LIN {X 0,Y 573.234,Z 422.71,A -85,B 0,C 180,E1 -2362.338,E2 -2362.338} C_VEL
LIN {X 0,Y 573.247,Z 422.704,A -85,B 0,C 180,E1 -2364.401,E2 -2364.401} C_VEL
LIN {X 0,Y 572.62,Z 422.786,A -85,B 0,C 180,E1 -2364.987,E2 -2364.987} C_VEL
LIN {X 0,Y 569.776,Z 423.137,A -85,B 0,C 180,E1 -2365.938,E2 -2365.938} C_VEL
LIN {X 0,Y 567.346,Z 423.44,A -85,B 0,C 180,E1 -2366.704,E2 -2366.704} C_VEL
LIN {X 0,Y 566.295,Z 423.569,A -85,B 0,C 180,E1 -2367.295,E2 -2367.295} C_VEL
LIN {X 0,Y 566.207,Z 423.58,A -85,B 0,C 180,E1 -2367.495,E2 -2367.495} C_VEL
LIN {X 0,Y 566.184,Z 423.588,A -85,B 0,C 180,E1 -2370.593,E2 -2370.593} C_VEL
LIN {X 0,Y 566.225,Z 423.58,A -85,B 0,C 180,E1 -2373.102,E2 -2373.102} C_VEL
LIN {X 0,Y 566.212,Z 423.583,A -85,B 0,C 180,E1 -2376.217,E2 -2376.217} C_VEL
LIN {X 0,Y 566.212,Z 423.58,A -85,B 0,C 180,E1 -2379.274,E2 -2379.274} C_VEL
LIN {X 0,Y 566.215,Z 423.58,A -85,B 0,C 180,E1 -2382.088,E2 -2382.088} C_VEL
LIN {X 0,Y 566.172,Z 423.584,A -85,B 0,C 180,E1 -2385.036,E2 -2385.036} C_VEL
LIN {X 0,Y 566.189,Z 423.583,A -85,B 0,C 180,E1 -2387.911,E2 -2387.911} C_VEL
LIN {X 0,Y 566.222,Z 423.579,A -85,B 0,C 180,E1 -2390.728,E2 -2390.728} C_VEL
LIN {X 0,Y 566.219,Z 423.582,A -85,B 0,C 180,E1 -2393.784,E2 -2393.784} C_VEL
LIN {X 0,Y 566.213,Z 423.581,A -85,B 0,C 180,E1 -2396.266,E2 -2396.266} C_VEL
LIN {X 0,Y 566.195,Z 423.582,A -85,B 0,C 180,E1 -2398.924,E2 -2398.924} C_VEL
LIN {X 0,Y 566.196,Z 423.584,A -85,B 0,C 180,E1 -2401.047,E2 -2401.047} C_VEL
LIN {X 0,Y 566.219,Z 423.582,A -85,B 0,C 180,E1 -2403.46,E2 -2403.46} C_VEL
LIN {X 0,Y 566.201,Z 423.582,A -85,B 0,C 180,E1 -2405.82,E2 -2405.82} C_VEL
LIN {X 0,Y 566.211,Z 423.583,A -85,B 0,C 180,E1 -2408.903,E2 -2408.903} C_VEL
LIN {X 0,Y 566.203,Z 423.581,A -85,B 0,C 180,E1 -2411.173,E2 -2411.173} C_VEL
LIN {X 0,Y 566.217,Z 423.582,A -85,B 0,C 180,E1 -2413.413,E2 -2413.413} C_VEL
LIN {X 0,Y 566.201,Z 423.581,A -85,B 0,C 180,E1 -2416.359,E2 -2416.359} C_VEL
LIN {X 0,Y 566.239,Z 423.58,A -85,B 0,C 180,E1 -2418.676,E2 -2418.676} C_VEL
LIN {X 0,Y 566.232,Z 423.582,A -85,B 0,C 180,E1 -2421.435,E2 -2421.435} C_VEL
LIN {X 0,Y 566.259,Z 423.577,A -85,B 0,C 180,E1 -2424.302,E2 -2424.302} C_VEL
LIN {X 0,Y 566.287,Z 423.572,A -85,B 0,C 180,E1 -2427.866,E2 -2427.866} C_VEL
LIN {X 0,Y 566.302,Z 423.569,A -85,B 0,C 180,E1 -2430.711,E2 -2430.711} C_VEL
LIN {X 0,Y 566.274,Z 423.573,A -85,B 0,C 180,E1 -2432.845,E2 -2432.845} C_VEL
LIN {X 0,Y 566.266,Z 423.573,A -85,B 0,C 180,E1 -2435.698,E2 -2435.698} C_VEL
LIN {X 0,Y 566.211,Z 423.58,A -85,B 0,C 180,E1 -2438.566,E2 -2438.566} C_VEL
LIN {X 0,Y 566.246,Z 423.576,A -85,B 0,C 180,E1 -2441.454,E2 -2441.454} C_VEL
LIN {X 0,Y 566.239,Z 423.578,A -85,B 0,C 180,E1 -2444.506,E2 -2444.506} C_VEL
LIN {X 0,Y 566.202,Z 423.584,A -85,B 0,C 180,E1 -2447.331,E2 -2447.331} C_VEL
LIN {X 0,Y 566.211,Z 423.584,A -85,B 0,C 180,E1 -2450.337,E2 -2450.337} C_VEL
LIN {X 0,Y 566.193,Z 423.583,A -85,B 0,C 180,E1 -2453.403,E2 -2453.403} C_VEL
LIN {X 0,Y 566.217,Z 423.583,A -85,B 0,C 180,E1 -2455.748,E2 -2455.748} C_VEL
LIN {X 0,Y 566.209,Z 423.581,A -85,B 0,C 180,E1 -2458.202,E2 -2458.202} C_VEL
LIN {X 0,Y 566.201,Z 423.584,A -85,B 0,C 180,E1 -2461.077,E2 -2461.077} C_VEL
LIN {X 0,Y 566.188,Z 423.585,A -85,B 0,C 180,E1 -2463.73,E2 -2463.73} C_VEL
LIN {X 0,Y 565.994,Z 423.636,A -85,B 0,C 180,E1 -2465.704,E2 -2465.704} C_VEL
LIN {X 0,Y 565.976,Z 426.477,A -85,B 0,C 180,E1 -2468.528,E2 -2468.528} C_VEL
LIN {X 0,Y 565.936,Z 429.152,A -85,B 0,C 180,E1 -2471.16,E2 -2471.16} C_VEL
LIN {X 0,Y 565.954,Z 432.13,A -85,B 0,C 180,E1 -2474.059,E2 -2474.059} C_VEL
LIN {X 0,Y 565.928,Z 435.2,A -85,B 0,C 180,E1 -2477.112,E2 -2477.112} C_VEL
LIN {X 0,Y 565.889,Z 438.183,A -85,B 0,C 180,E1 -2479.773,E2 -2479.773} C_VEL
LIN {X 0,Y 565.844,Z 441.501,A -85,B 0,C 180,E1 -2482.645,E2 -2482.645} C_VEL
LIN {X 0,Y 565.859,Z 444.449,A -85,B 0,C 180,E1 -2485.157,E2 -2485.157} C_VEL
LIN {X 0,Y 565.879,Z 446.388,A -85,B 0,C 180,E1 -2486.791,E2 -2486.791} C_VEL
LIN {X 0,Y 567.394,Z 454.471,A -85,B 0,C 180,E1 -2486.992,E2 -2486.992} C_VEL
LIN {X 0,Y 567.255,Z 468.399,A -85,B 0,C 180,E1 -2487.361,E2 -2487.361} C_VEL
LIN {X 0,Y 567.079,Z 481.532,A -85,B 0,C 180,E1 -2487.85,E2 -2487.85} C_VEL
LIN {X 0,Y 566.886,Z 495.141,A -85,B 0,C 180,E1 -2488.517,E2 -2488.517} C_VEL
LIN {X 0,Y 566.716,Z 507.038,A -85,B 0,C 180,E1 -2489.251,E2 -2489.251} C_VEL
LIN {X 0,Y 566.534,Z 518.876,A -85,B 0,C 180,E1 -2490.148,E2 -2490.148} C_VEL
LIN {X 0,Y 566.38,Z 528.827,A -85,B 0,C 180,E1 -2491.057,E2 -2491.057} C_VEL
LIN {X 0,Y 566.217,Z 538.024,A -85,B 0,C 180,E1 -2492.059,E2 -2492.059} C_VEL
LIN {X 0,Y 566.123,Z 547.123,A -85,B 0,C 180,E1 -2493.256,E2 -2493.256} C_VEL
LIN {X 0,Y 566.004,Z 554.487,A -85,B 0,C 180,E1 -2494.438,E2 -2494.438} C_VEL
LIN {X 0,Y 565.951,Z 561.337,A -85,B 0,C 180,E1 -2495.808,E2 -2495.808} C_VEL
LIN {X 0,Y 565.93,Z 565.213,A -85,B 0,C 180,E1 -2496.773,E2 -2496.773} C_VEL
LIN {X 0,Y 565.88,Z 569.42,A -85,B 0,C 180,E1 -2498.124,E2 -2498.124} C_VEL
LIN {X 0,Y 565.891,Z 571.213,A -85,B 0,C 180,E1 -2498.89,E2 -2498.89} C_VEL
LIN {X 0,Y 565.832,Z 573.597,A -85,B 0,C 180,E1 -2500.406,E2 -2500.406} C_VEL
LIN {X 0,Y 565.83,Z 574.477,A -85,B 0,C 180,E1 -2501.909,E2 -2501.909} C_VEL
LIN {X 0,Y 565.841,Z 573.9,A -85,B 0,C 180,E1 -2503.401,E2 -2503.401} C_VEL
LIN {X 0,Y 565.84,Z 571.856,A -85,B 0,C 180,E1 -2504.88,E2 -2504.88} C_VEL
LIN {X 0,Y 565.899,Z 568.345,A -85,B 0,C 180,E1 -2506.351,E2 -2506.351} C_VEL
LIN {X 0,Y 565.941,Z 563.307,A -85,B 0,C 180,E1 -2507.812,E2 -2507.812} C_VEL
LIN {X 0,Y 565.973,Z 558.307,A -85,B 0,C 180,E1 -2508.93,E2 -2508.93} C_VEL
LIN {X 0,Y 566.075,Z 551.435,A -85,B 0,C 180,E1 -2510.171,E2 -2510.171} C_VEL
LIN {X 0,Y 566.125,Z 542.804,A -85,B 0,C 180,E1 -2511.433,E2 -2511.433} C_VEL
LIN {X 0,Y 566.313,Z 533.799,A -85,B 0,C 180,E1 -2512.513,E2 -2512.513} C_VEL
LIN {X 0,Y 566.448,Z 522.985,A -85,B 0,C 180,E1 -2513.589,E2 -2513.589} C_VEL
LIN {X 0,Y 566.645,Z 512.043,A -85,B 0,C 180,E1 -2514.484,E2 -2514.484} C_VEL
LIN {X 0,Y 566.779,Z 500.105,A -85,B 0,C 180,E1 -2515.288,E2 -2515.288} C_VEL
LIN {X 0,Y 567.003,Z 486.787,A -85,B 0,C 180,E1 -2516.002,E2 -2516.002} C_VEL
LIN {X 0,Y 567.196,Z 473.978,A -85,B 0,C 180,E1 -2516.537,E2 -2516.537} C_VEL
LIN {X 0,Y 567.341,Z 460.316,A -85,B 0,C 180,E1 -2516.96,E2 -2516.96} C_VEL
LIN {X 0,Y 567.167,Z 452.884,A -85,B 0,C 180,E1 -2517.137,E2 -2517.137} C_VEL
LIN {X 0,Y 565.851,Z 446.378,A -85,B 0,C 180,E1 -2517.308,E2 -2517.308} C_VEL
LIN {X 0,Y 565.889,Z 443.19,A -85,B 0,C 180,E1 -2520,E2 -2520} C_VEL
LIN {X 0,Y 565.883,Z 439.872,A -85,B 0,C 180,E1 -2522.847,E2 -2522.847} C_VEL
LIN {X 0,Y 565.959,Z 436.605,A -85,B 0,C 180,E1 -2525.701,E2 -2525.701} C_VEL
LIN {X 0,Y 565.979,Z 434.458,A -85,B 0,C 180,E1 -2527.851,E2 -2527.851} C_VEL
LIN {X 0,Y 566.06,Z 431.516,A -85,B 0,C 180,E1 -2531.241,E2 -2531.241} C_VEL
LIN {X 0,Y 566.065,Z 428.336,A -85,B 0,C 180,E1 -2534.443,E2 -2534.443} C_VEL
LIN {X 0,Y 566.096,Z 425.665,A -85,B 0,C 180,E1 -2537.335,E2 -2537.335} C_VEL
LIN {X 0,Y 566.111,Z 423.597,A -85,B 0,C 180,E1 -2539.584,E2 -2539.584} C_VEL
LIN {X 0,Y 566.191,Z 423.584,A -85,B 0,C 180,E1 -2541.863,E2 -2541.863} C_VEL
LIN {X 0,Y 566.229,Z 423.575,A -85,B 0,C 180,E1 -2544.961,E2 -2544.961} C_VEL
LIN {X 0,Y 566.219,Z 423.576,A -85,B 0,C 180,E1 -2547.339,E2 -2547.339} C_VEL
LIN {X 0,Y 566.222,Z 423.58,A -85,B 0,C 180,E1 -2549.768,E2 -2549.768} C_VEL
LIN {X 0,Y 566.204,Z 423.581,A -85,B 0,C 180,E1 -2552.431,E2 -2552.431} C_VEL
LIN {X 0,Y 566.208,Z 423.577,A -85,B 0,C 180,E1 -2554.995,E2 -2554.995} C_VEL
LIN {X 0,Y 566.192,Z 423.581,A -85,B 0,C 180,E1 -2557.461,E2 -2557.461} C_VEL
LIN {X 0,Y 566.223,Z 423.581,A -85,B 0,C 180,E1 -2560.198,E2 -2560.198} C_VEL
LIN {X 0,Y 566.202,Z 423.579,A -85,B 0,C 180,E1 -2563.054,E2 -2563.054} C_VEL
LIN {X 0,Y 566.199,Z 423.587,A -85,B 0,C 180,E1 -2566.049,E2 -2566.049} C_VEL
LIN {X 0,Y 566.209,Z 423.582,A -85,B 0,C 180,E1 -2568.864,E2 -2568.864} C_VEL
LIN {X 0,Y 566.262,Z 423.679,A -85,B 0,C 180,E1 -2569.587,E2 -2569.587} C_VEL
LIN {X 0,Y 566.891,Z 427.712,A -85,B 0,C 180,E1 -2571.356,E2 -2571.356} C_VEL
LIN {X 0,Y 566.768,Z 433.908,A -85,B 0,C 180,E1 -2573.708,E2 -2573.708} C_VEL
LIN {X 0,Y 566.619,Z 441.021,A -85,B 0,C 180,E1 -2576.204,E2 -2576.204} C_VEL
LIN {X 0,Y 566.57,Z 449.293,A -85,B 0,C 180,E1 -2578.86,E2 -2578.86} C_VEL
LIN {X 0,Y 566.478,Z 459.198,A -85,B 0,C 180,E1 -2581.872,E2 -2581.872} C_VEL
LIN {X 0,Y 566.392,Z 468.297,A -85,B 0,C 180,E1 -2584.639,E2 -2584.639} C_VEL
LIN {X 0,Y 566.27,Z 477.307,A -85,B 0,C 180,E1 -2587.373,E2 -2587.373} C_VEL
LIN {X 0,Y 566.193,Z 487.546,A -85,B 0,C 180,E1 -2590.419,E2 -2590.419} C_VEL
LIN {X 0,Y 566.11,Z 497.786,A -85,B 0,C 180,E1 -2593.41,E2 -2593.41} C_VEL
LIN {X 0,Y 566.085,Z 502.186,A -85,B 0,C 180,E1 -2594.68,E2 -2594.68} C_VEL
LIN {X 0,Y 567.44,Z 510.182,A -85,B 0,C 180,E1 -2594.861,E2 -2594.861} C_VEL
LIN {X 0,Y 567.305,Z 524.025,A -85,B 0,C 180,E1 -2595.185,E2 -2595.185} C_VEL
LIN {X 0,Y 567.112,Z 537.717,A -85,B 0,C 180,E1 -2595.65,E2 -2595.65} C_VEL
LIN {X 0,Y 566.975,Z 551.647,A -85,B 0,C 180,E1 -2596.287,E2 -2596.287} C_VEL
LIN {X 0,Y 566.763,Z 564.104,A -85,B 0,C 180,E1 -2597.012,E2 -2597.012} C_VEL
LIN {X 0,Y 566.576,Z 576.643,A -85,B 0,C 180,E1 -2597.918,E2 -2597.918} C_VEL
LIN {X 0,Y 566.446,Z 587.32,A -85,B 0,C 180,E1 -2598.861,E2 -2598.861} C_VEL
LIN {X 0,Y 566.206,Z 597.853,A -85,B 0,C 180,E1 -2599.993,E2 -2599.993} C_VEL
LIN {X 0,Y 566.132,Z 606.173,A -85,B 0,C 180,E1 -2601.073,E2 -2601.073} C_VEL
LIN {X 0,Y 566.046,Z 614.128,A -85,B 0,C 180,E1 -2602.33,E2 -2602.33} C_VEL
LIN {X 0,Y 565.943,Z 620.528,A -85,B 0,C 180,E1 -2603.583,E2 -2603.583} C_VEL
LIN {X 0,Y 565.928,Z 624.961,A -85,B 0,C 180,E1 -2604.656,E2 -2604.656} C_VEL
LIN {X 0,Y 565.956,Z 628.443,A -85,B 0,C 180,E1 -2605.727,E2 -2605.727} C_VEL
LIN {X 0,Y 565.874,Z 631.832,A -85,B 0,C 180,E1 -2607.152,E2 -2607.152} C_VEL
LIN {X 0,Y 565.84,Z 633.833,A -85,B 0,C 180,E1 -2608.577,E2 -2608.577} C_VEL
LIN {X 0,Y 565.837,Z 634.5,A -85,B 0,C 180,E1 -2610,E2 -2610} C_VEL
LIN {X 0,Y 565.84,Z 633.833,A -85,B 0,C 180,E1 -2611.423,E2 -2611.423} C_VEL
LIN {X 0,Y 565.874,Z 631.834,A -85,B 0,C 180,E1 -2612.848,E2 -2612.848} C_VEL
LIN {X 0,Y 565.956,Z 628.445,A -85,B 0,C 180,E1 -2614.273,E2 -2614.273} C_VEL
LIN {X 0,Y 565.988,Z 623.568,A -85,B 0,C 180,E1 -2615.701,E2 -2615.701} C_VEL
LIN {X 0,Y 565.992,Z 619.045,A -85,B 0,C 180,E1 -2616.739,E2 -2616.739} C_VEL
LIN {X 0,Y 566.047,Z 612.038,A -85,B 0,C 180,E1 -2618.029,E2 -2618.029} C_VEL
LIN {X 0,Y 566.177,Z 603.56,A -85,B 0,C 180,E1 -2619.286,E2 -2619.286} C_VEL
LIN {X 0,Y 566.294,Z 594.709,A -85,B 0,C 180,E1 -2620.367,E2 -2620.367} C_VEL
LIN {X 0,Y 566.485,Z 583.993,A -85,B 0,C 180,E1 -2621.449,E2 -2621.449} C_VEL
LIN {X 0,Y 566.638,Z 573.145,A -85,B 0,C 180,E1 -2622.354,E2 -2622.354} C_VEL
LIN {X 0,Y 566.774,Z 561.262,A -85,B 0,C 180,E1 -2623.17,E2 -2623.17} C_VEL
LIN {X 0,Y 567.046,Z 548.1,A -85,B 0,C 180,E1 -2623.894,E2 -2623.894} C_VEL
LIN {X 0,Y 567.194,Z 535.146,A -85,B 0,C 180,E1 -2624.45,E2 -2624.45} C_VEL
LIN {X 0,Y 567.335,Z 520.935,A -85,B 0,C 180,E1 -2624.899,E2 -2624.899} C_VEL
LIN {X 0,Y 567.341,Z 508.652,A -85,B 0,C 180,E1 -2625.17,E2 -2625.17} C_VEL
LIN {X 0,Y 566.086,Z 502.186,A -85,B 0,C 180,E1 -2625.32,E2 -2625.32} C_VEL
LIN {X 0,Y 566.15,Z 492.666,A -85,B 0,C 180,E1 -2628.079,E2 -2628.079} C_VEL
LIN {X 0,Y 566.215,Z 483.706,A -85,B 0,C 180,E1 -2630.716,E2 -2630.716} C_VEL
LIN {X 0,Y 566.312,Z 474.747,A -85,B 0,C 180,E1 -2633.398,E2 -2633.398} C_VEL
LIN {X 0,Y 566.406,Z 465.778,A -85,B 0,C 180,E1 -2636.134,E2 -2636.134} C_VEL
LIN {X 0,Y 566.502,Z 456.675,A -85,B 0,C 180,E1 -2638.935,E2 -2638.935} C_VEL
LIN {X 0,Y 566.607,Z 447.555,A -85,B 0,C 180,E1 -2641.813,E2 -2641.813} C_VEL
LIN {X 0,Y 566.777,Z 438.577,A -85,B 0,C 180,E1 -2644.777,E2 -2644.777} C_VEL
LIN {X 0,Y 566.892,Z 430.796,A -85,B 0,C 180,E1 -2647.492,E2 -2647.492} C_VEL
LIN {X 0,Y 566.907,Z 427.604,A -85,B 0,C 180,E1 -2648.646,E2 -2648.646} C_VEL
LIN {X 0,Y 566.223,Z 423.582,A -85,B 0,C 180,E1 -2650.252,E2 -2650.252} C_VEL
LIN {X 0,Y 566.198,Z 423.583,A -85,B 0,C 180,E1 -2653.053,E2 -2653.053} C_VEL
LIN {X 0,Y 566.199,Z 423.583,A -85,B 0,C 180,E1 -2656.048,E2 -2656.048} C_VEL
LIN {X 0,Y 566.208,Z 423.582,A -85,B 0,C 180,E1 -2658.863,E2 -2658.863} C_VEL
LIN {X 0,Y 566.186,Z 423.586,A -85,B 0,C 180,E1 -2661.637,E2 -2661.637} C_VEL
LIN {X 0,Y 566.191,Z 423.584,A -85,B 0,C 180,E1 -2664.31,E2 -2664.31} C_VEL
LIN {X 0,Y 566.224,Z 423.579,A -85,B 0,C 180,E1 -2666.898,E2 -2666.898} C_VEL
LIN {X 0,Y 566.189,Z 423.583,A -85,B 0,C 180,E1 -2669.408,E2 -2669.408} C_VEL
LIN {X 0,Y 566.222,Z 423.579,A -85,B 0,C 180,E1 -2671.858,E2 -2671.858} C_VEL
LIN {X 0,Y 566.222,Z 423.583,A -85,B 0,C 180,E1 -2674.251,E2 -2674.251} C_VEL
LIN {X 0,Y 566.185,Z 423.585,A -85,B 0,C 180,E1 -2676.713,E2 -2676.713} C_VEL
LIN {X 0,Y 566.214,Z 423.584,A -85,B 0,C 180,E1 -2679.663,E2 -2679.663} C_VEL
LIN {X 0,Y 566.198,Z 423.585,A -85,B 0,C 180,E1 -2682.668,E2 -2682.668} C_VEL
LIN {X 0,Y 566.227,Z 423.579,A -85,B 0,C 180,E1 -2685.627,E2 -2685.627} C_VEL
LIN {X 0,Y 566.268,Z 423.573,A -85,B 0,C 180,E1 -2688.654,E2 -2688.654} C_VEL
LIN {X 0,Y 566.243,Z 423.576,A -85,B 0,C 180,E1 -2691.435,E2 -2691.435} C_VEL
LIN {X 0,Y 566.257,Z 423.575,A -85,B 0,C 180,E1 -2694.302,E2 -2694.302} C_VEL
LIN {X 0,Y 566.275,Z 423.574,A -85,B 0,C 180,E1 -2697.866,E2 -2697.866} C_VEL
LIN {X 0,Y 566.299,Z 423.57,A -85,B 0,C 180,E1 -2700.711,E2 -2700.711} C_VEL
LIN {X 0,Y 566.274,Z 423.574,A -85,B 0,C 180,E1 -2702.846,E2 -2702.846} C_VEL
LIN {X 0,Y 566.266,Z 423.576,A -85,B 0,C 180,E1 -2705.698,E2 -2705.698} C_VEL
LIN {X 0,Y 566.242,Z 423.581,A -85,B 0,C 180,E1 -2708.566,E2 -2708.566} C_VEL
LIN {X 0,Y 566.235,Z 423.581,A -85,B 0,C 180,E1 -2711.455,E2 -2711.455} C_VEL
LIN {X 0,Y 566.227,Z 423.579,A -85,B 0,C 180,E1 -2714.507,E2 -2714.507} C_VEL
LIN {X 0,Y 566.199,Z 423.582,A -85,B 0,C 180,E1 -2717.332,E2 -2717.332} C_VEL
LIN {X 0,Y 566.215,Z 423.58,A -85,B 0,C 180,E1 -2720.337,E2 -2720.337} C_VEL
LIN {X 0,Y 566.185,Z 423.585,A -85,B 0,C 180,E1 -2723.404,E2 -2723.404} C_VEL
LIN {X 0,Y 566.21,Z 423.58,A -85,B 0,C 180,E1 -2725.749,E2 -2725.749} C_VEL
LIN {X 0,Y 566.207,Z 423.58,A -85,B 0,C 180,E1 -2727.495,E2 -2727.495} C_VEL
LIN {X 0,Y 565.531,Z 423.667,A -85,B 0,C 180,E1 -2728.089,E2 -2728.089} C_VEL
LIN {X 0,Y 562.662,Z 424.025,A -85,B 0,C 180,E1 -2729.052,E2 -2729.052} C_VEL
LIN {X 0,Y 560.248,Z 424.324,A -85,B 0,C 180,E1 -2729.828,E2 -2729.828} C_VEL
LIN {X 0,Y 559.22,Z 424.454,A -85,B 0,C 180,E1 -2730.427,E2 -2730.427} C_VEL
LIN {X 0,Y 559.141,Z 424.459,A -85,B 0,C 180,E1 -2730.629,E2 -2730.629} C_VEL
LIN {X 0,Y 559.161,Z 424.461,A -85,B 0,C 180,E1 -2733.575,E2 -2733.575} C_VEL
LIN {X 0,Y 559.164,Z 424.459,A -85,B 0,C 180,E1 -2736.449,E2 -2736.449} C_VEL
LIN {X 0,Y 559.172,Z 424.46,A -85,B 0,C 180,E1 -2738.935,E2 -2738.935} C_VEL
LIN {X 0,Y 559.178,Z 424.457,A -85,B 0,C 180,E1 -2742.138,E2 -2742.138} C_VEL
LIN {X 0,Y 559.139,Z 424.461,A -85,B 0,C 180,E1 -2744.74,E2 -2744.74} C_VEL
LIN {X 0,Y 559.159,Z 424.462,A -85,B 0,C 180,E1 -2747.257,E2 -2747.257} C_VEL
LIN {X 0,Y 559.185,Z 424.457,A -85,B 0,C 180,E1 -2750.136,E2 -2750.136} C_VEL
LIN {X 0,Y 559.147,Z 424.461,A -85,B 0,C 180,E1 -2752.893,E2 -2752.893} C_VEL
LIN {X 0,Y 559.159,Z 424.461,A -85,B 0,C 180,E1 -2755.557,E2 -2755.557} C_VEL
LIN {X 0,Y 559.167,Z 424.461,A -85,B 0,C 180,E1 -2758.138,E2 -2758.138} C_VEL
LIN {X 0,Y 559.159,Z 424.462,A -85,B 0,C 180,E1 -2760.648,E2 -2760.648} C_VEL
LIN {X 0,Y 559.173,Z 424.457,A -85,B 0,C 180,E1 -2763.173,E2 -2763.173} C_VEL
LIN {X 0,Y 559.159,Z 424.459,A -85,B 0,C 180,E1 -2765.495,E2 -2765.495} C_VEL
LIN {X 0,Y 559.175,Z 424.457,A -85,B 0,C 180,E1 -2768.624,E2 -2768.624} C_VEL
LIN {X 0,Y 559.166,Z 424.458,A -85,B 0,C 180,E1 -2770.927,E2 -2770.927} C_VEL
LIN {X 0,Y 559.169,Z 424.458,A -85,B 0,C 180,E1 -2773.948,E2 -2773.948} C_VEL
LIN {X 0,Y 559.176,Z 424.458,A -85,B 0,C 180,E1 -2776.184,E2 -2776.184} C_VEL
LIN {X 0,Y 559.198,Z 424.454,A -85,B 0,C 180,E1 -2779.134,E2 -2779.134} C_VEL
LIN {X 0,Y 559.209,Z 424.452,A -85,B 0,C 180,E1 -2782.054,E2 -2782.054} C_VEL
LIN {X 0,Y 559.255,Z 424.447,A -85,B 0,C 180,E1 -2784.953,E2 -2784.953} C_VEL
LIN {X 0,Y 559.258,Z 424.447,A -85,B 0,C 180,E1 -2787.839,E2 -2787.839} C_VEL
LIN {X 0,Y 559.273,Z 424.445,A -85,B 0,C 180,E1 -2790.72,E2 -2790.72} C_VEL
LIN {X 0,Y 559.241,Z 424.449,A -85,B 0,C 180,E1 -2792.881,E2 -2792.881} C_VEL
LIN {X 0,Y 559.236,Z 424.449,A -85,B 0,C 180,E1 -2795.77,E2 -2795.77} C_VEL
LIN {X 0,Y 559.176,Z 424.456,A -85,B 0,C 180,E1 -2798.674,E2 -2798.674} C_VEL
LIN {X 0,Y 559.21,Z 424.453,A -85,B 0,C 180,E1 -2801.6,E2 -2801.6} C_VEL
LIN {X 0,Y 559.204,Z 424.455,A -85,B 0,C 180,E1 -2804.595,E2 -2804.595} C_VEL
LIN {X 0,Y 559.161,Z 424.462,A -85,B 0,C 180,E1 -2807.557,E2 -2807.557} C_VEL
LIN {X 0,Y 559.169,Z 424.458,A -85,B 0,C 180,E1 -2809.837,E2 -2809.837} C_VEL
LIN {X 0,Y 559.144,Z 424.461,A -85,B 0,C 180,E1 -2812.152,E2 -2812.152} C_VEL
LIN {X 0,Y 559.182,Z 424.456,A -85,B 0,C 180,E1 -2815.186,E2 -2815.186} C_VEL
LIN {X 0,Y 559.194,Z 424.454,A -85,B 0,C 180,E1 -2817.711,E2 -2817.711} C_VEL
LIN {X 0,Y 559.165,Z 424.46,A -85,B 0,C 180,E1 -2821.018,E2 -2821.018} C_VEL
LIN {X 0,Y 559.137,Z 424.465,A -85,B 0,C 180,E1 -2823.944,E2 -2823.944} C_VEL
LIN {X 0,Y 558.938,Z 424.78,A -85,B 0,C 180,E1 -2826.225,E2 -2826.225} C_VEL
LIN {X 0,Y 558.884,Z 427.524,A -85,B 0,C 180,E1 -2828.957,E2 -2828.957} C_VEL
LIN {X 0,Y 558.869,Z 430.384,A -85,B 0,C 180,E1 -2831.796,E2 -2831.796} C_VEL
LIN {X 0,Y 558.863,Z 432.807,A -85,B 0,C 180,E1 -2834.208,E2 -2834.208} C_VEL
LIN {X 0,Y 558.857,Z 435.877,A -85,B 0,C 180,E1 -2837.227,E2 -2837.227} C_VEL
LIN {X 0,Y 558.799,Z 438.89,A -85,B 0,C 180,E1 -2840.101,E2 -2840.101} C_VEL
LIN {X 0,Y 558.742,Z 442.044,A -85,B 0,C 180,E1 -2842.86,E2 -2842.86} C_VEL
LIN {X 0,Y 558.753,Z 445.14,A -85,B 0,C 180,E1 -2845.527,E2 -2845.527} C_VEL
LIN {X 0,Y 558.781,Z 446.466,A -85,B 0,C 180,E1 -2846.603,E2 -2846.603} C_VEL
LIN {X 0,Y 560.503,Z 455.736,A -85,B 0,C 180,E1 -2846.829,E2 -2846.829} C_VEL
LIN {X 0,Y 560.367,Z 469.38,A -85,B 0,C 180,E1 -2847.209,E2 -2847.209} C_VEL
LIN {X 0,Y 560.17,Z 482.707,A -85,B 0,C 180,E1 -2847.724,E2 -2847.724} C_VEL
LIN {X 0,Y 559.965,Z 495.641,A -85,B 0,C 180,E1 -2848.375,E2 -2848.375} C_VEL
LIN {X 0,Y 559.757,Z 507.504,A -85,B 0,C 180,E1 -2849.122,E2 -2849.122} C_VEL
LIN {X 0,Y 559.52,Z 519.785,A -85,B 0,C 180,E1 -2850.075,E2 -2850.075} C_VEL
LIN {X 0,Y 559.354,Z 530.312,A -85,B 0,C 180,E1 -2851.07,E2 -2851.07} C_VEL
LIN {X 0,Y 559.143,Z 539.25,A -85,B 0,C 180,E1 -2852.082,E2 -2852.082} C_VEL
LIN {X 0,Y 559.053,Z 547.463,A -85,B 0,C 180,E1 -2853.195,E2 -2853.195} C_VEL
LIN {X 0,Y 558.932,Z 555.313,A -85,B 0,C 180,E1 -2854.49,E2 -2854.49} C_VEL
LIN {X 0,Y 558.872,Z 561.995,A -85,B 0,C 180,E1 -2855.877,E2 -2855.877} C_VEL
LIN {X 0,Y 558.816,Z 566.402,A -85,B 0,C 180,E1 -2857.053,E2 -2857.053} C_VEL
LIN {X 0,Y 558.798,Z 570.568,A -85,B 0,C 180,E1 -2858.541,E2 -2858.541} C_VEL
LIN {X 0,Y 558.757,Z 572.226,A -85,B 0,C 180,E1 -2859.379,E2 -2859.379} C_VEL
LIN {X 0,Y 558.77,Z 574.065,A -85,B 0,C 180,E1 -2860.912,E2 -2860.912} C_VEL
LIN {X 0,Y 558.739,Z 574.423,A -85,B 0,C 180,E1 -2862.429,E2 -2862.429} C_VEL
LIN {X 0,Y 558.735,Z 573.342,A -85,B 0,C 180,E1 -2863.935,E2 -2863.935} C_VEL
LIN {X 0,Y 558.776,Z 570.828,A -85,B 0,C 180,E1 -2865.431,E2 -2865.431} C_VEL
LIN {X 0,Y 558.812,Z 566.815,A -85,B 0,C 180,E1 -2866.916,E2 -2866.916} C_VEL
LIN {X 0,Y 558.867,Z 562.762,A -85,B 0,C 180,E1 -2868.024,E2 -2868.024} C_VEL
LIN {X 0,Y 558.926,Z 557.755,A -85,B 0,C 180,E1 -2869.128,E2 -2869.128} C_VEL
LIN {X 0,Y 559.013,Z 550.596,A -85,B 0,C 180,E1 -2870.411,E2 -2870.411} C_VEL
LIN {X 0,Y 559.087,Z 543.145,A -85,B 0,C 180,E1 -2871.506,E2 -2871.506} C_VEL
LIN {X 0,Y 559.29,Z 534.207,A -85,B 0,C 180,E1 -2872.6,E2 -2872.6} C_VEL
LIN {X 0,Y 559.452,Z 523.47,A -85,B 0,C 180,E1 -2873.689,E2 -2873.689} C_VEL
LIN {X 0,Y 559.654,Z 512.632,A -85,B 0,C 180,E1 -2874.596,E2 -2874.596} C_VEL
LIN {X 0,Y 559.841,Z 500.822,A -85,B 0,C 180,E1 -2875.41,E2 -2875.41} C_VEL
LIN {X 0,Y 560.07,Z 487.76,A -85,B 0,C 180,E1 -2876.132,E2 -2876.132} C_VEL
LIN {X 0,Y 560.315,Z 473.967,A -85,B 0,C 180,E1 -2876.719,E2 -2876.719} C_VEL
LIN {X 0,Y 560.488,Z 460.279,A -85,B 0,C 180,E1 -2877.147,E2 -2877.147} C_VEL
LIN {X 0,Y 560.293,Z 453.983,A -85,B 0,C 180,E1 -2877.304,E2 -2877.304} C_VEL
LIN {X 0,Y 558.747,Z 446.387,A -85,B 0,C 180,E1 -2877.499,E2 -2877.499} C_VEL
LIN {X 0,Y 558.795,Z 443.464,A -85,B 0,C 180,E1 -2880,E2 -2880} C_VEL
LIN {X 0,Y 558.805,Z 440.145,A -85,B 0,C 180,E1 -2882.883,E2 -2882.883} C_VEL
LIN {X 0,Y 558.817,Z 437.702,A -85,B 0,C 180,E1 -2885.05,E2 -2885.05} C_VEL
LIN {X 0,Y 558.905,Z 435.733,A -85,B 0,C 180,E1 -2887.224,E2 -2887.224} C_VEL
LIN {X 0,Y 558.956,Z 433.227,A -85,B 0,C 180,E1 -2890.138,E2 -2890.138} C_VEL
LIN {X 0,Y 558.949,Z 431.042,A -85,B 0,C 180,E1 -2892.342,E2 -2892.342} C_VEL
LIN {X 0,Y 559.01,Z 428.378,A -85,B 0,C 180,E1 -2895.308,E2 -2895.308} C_VEL
LIN {X 0,Y 559.037,Z 426.215,A -85,B 0,C 180,E1 -2897.561,E2 -2897.561} C_VEL
LIN {X 0,Y 559.068,Z 424.475,A -85,B 0,C 180,E1 -2899.472,E2 -2899.472} C_VEL
LIN {X 0,Y 559.137,Z 424.466,A -85,B 0,C 180,E1 -2902.153,E2 -2902.153} C_VEL
LIN {X 0,Y 559.173,Z 424.453,A -85,B 0,C 180,E1 -2905.188,E2 -2905.188} C_VEL
LIN {X 0,Y 559.189,Z 424.455,A -85,B 0,C 180,E1 -2907.712,E2 -2907.712} C_VEL
LIN {X 0,Y 559.163,Z 424.462,A -85,B 0,C 180,E1 -2910.182,E2 -2910.182} C_VEL
LIN {X 0,Y 559.171,Z 424.455,A -85,B 0,C 180,E1 -2912.714,E2 -2912.714} C_VEL
LIN {X 0,Y 559.152,Z 424.457,A -85,B 0,C 180,E1 -2915.322,E2 -2915.322} C_VEL
LIN {X 0,Y 559.131,Z 424.467,A -85,B 0,C 180,E1 -2918.018,E2 -2918.018} C_VEL
LIN {X 0,Y 559.172,Z 424.454,A -85,B 0,C 180,E1 -2920.811,E2 -2920.811} C_VEL
LIN {X 0,Y 559.159,Z 424.463,A -85,B 0,C 180,E1 -2923.732,E2 -2923.732} C_VEL
LIN {X 0,Y 559.165,Z 424.458,A -85,B 0,C 180,E1 -2926.802,E2 -2926.802} C_VEL
LIN {X 0,Y 559.221,Z 424.628,A -85,B 0,C 180,E1 -2929.306,E2 -2929.306} C_VEL
LIN {X 0,Y 559.949,Z 429.783,A -85,B 0,C 180,E1 -2931.591,E2 -2931.591} C_VEL
LIN {X 0,Y 559.775,Z 435.607,A -85,B 0,C 180,E1 -2933.838,E2 -2933.838} C_VEL
LIN {X 0,Y 559.593,Z 443.021,A -85,B 0,C 180,E1 -2936.455,E2 -2936.455} C_VEL
LIN {X 0,Y 559.55,Z 449.656,A -85,B 0,C 180,E1 -2938.659,E2 -2938.659} C_VEL
LIN {X 0,Y 559.441,Z 459.079,A -85,B 0,C 180,E1 -2941.567,E2 -2941.567} C_VEL
LIN {X 0,Y 559.358,Z 468.143,A -85,B 0,C 180,E1 -2944.312,E2 -2944.312} C_VEL
LIN {X 0,Y 559.244,Z 477.307,A -85,B 0,C 180,E1 -2947.072,E2 -2947.072} C_VEL
LIN {X 0,Y 559.168,Z 487.546,A -85,B 0,C 180,E1 -2950.163,E2 -2950.163} C_VEL
LIN {X 0,Y 559.047,Z 497.786,A -85,B 0,C 180,E1 -2953.194,E2 -2953.194} C_VEL
LIN {X 0,Y 559.004,Z 502.186,A -85,B 0,C 180,E1 -2954.481,E2 -2954.481} C_VEL
LIN {X 0,Y 560.578,Z 511.037,A -85,B 0,C 180,E1 -2954.689,E2 -2954.689} C_VEL
LIN {X 0,Y 560.391,Z 525.746,A -85,B 0,C 180,E1 -2955.051,E2 -2955.051} C_VEL
LIN {X 0,Y 560.214,Z 539.97,A -85,B 0,C 180,E1 -2955.562,E2 -2955.562} C_VEL
LIN {X 0,Y 560.021,Z 553.398,A -85,B 0,C 180,E1 -2956.206,E2 -2956.206} C_VEL
LIN {X 0,Y 559.788,Z 565.517,A -85,B 0,C 180,E1 -2956.939,E2 -2956.939} C_VEL
LIN {X 0,Y 559.562,Z 577.754,A -85,B 0,C 180,E1 -2957.856,E2 -2957.856} C_VEL
LIN {X 0,Y 559.413,Z 588.777,A -85,B 0,C 180,E1 -2958.868,E2 -2958.868} C_VEL
LIN {X 0,Y 559.169,Z 599.34,A -85,B 0,C 180,E1 -2960.048,E2 -2960.048} C_VEL
LIN {X 0,Y 559.078,Z 607.409,A -85,B 0,C 180,E1 -2961.142,E2 -2961.142} C_VEL
LIN {X 0,Y 558.965,Z 615.136,A -85,B 0,C 180,E1 -2962.414,E2 -2962.414} C_VEL
LIN {X 0,Y 558.872,Z 620.528,A -85,B 0,C 180,E1 -2963.502,E2 -2963.502} C_VEL
LIN {X 0,Y 558.859,Z 624.961,A -85,B 0,C 180,E1 -2964.588,E2 -2964.588} C_VEL
LIN {X 0,Y 558.865,Z 628.443,A -85,B 0,C 180,E1 -2965.673,E2 -2965.673} C_VEL
LIN {X 0,Y 558.796,Z 631.832,A -85,B 0,C 180,E1 -2967.116,E2 -2967.116} C_VEL
LIN {X 0,Y 558.74,Z 633.833,A -85,B 0,C 180,E1 -2968.559,E2 -2968.559} C_VEL
LIN {X 0,Y 558.738,Z 634.5,A -85,B 0,C 180,E1 -2970,E2 -2970} C_VEL
LIN {X 0,Y 558.74,Z 633.834,A -85,B 0,C 180,E1 -2971.441,E2 -2971.441} C_VEL
LIN {X 0,Y 558.796,Z 631.834,A -85,B 0,C 180,E1 -2972.884,E2 -2972.884} C_VEL
LIN {X 0,Y 558.865,Z 628.445,A -85,B 0,C 180,E1 -2974.327,E2 -2974.327} C_VEL
LIN {X 0,Y 558.917,Z 623.568,A -85,B 0,C 180,E1 -2975.773,E2 -2975.773} C_VEL
LIN {X 0,Y 558.906,Z 617.054,A -85,B 0,C 180,E1 -2977.224,E2 -2977.224} C_VEL
LIN {X 0,Y 559.028,Z 609.802,A -85,B 0,C 180,E1 -2978.495,E2 -2978.495} C_VEL
LIN {X 0,Y 559.146,Z 600.824,A -85,B 0,C 180,E1 -2979.769,E2 -2979.769} C_VEL
LIN {X 0,Y 559.35,Z 591.394,A -85,B 0,C 180,E1 -2980.863,E2 -2980.863} C_VEL
LIN {X 0,Y 559.518,Z 580.953,A -85,B 0,C 180,E1 -2981.869,E2 -2981.869} C_VEL
LIN {X 0,Y 559.716,Z 569.438,A -85,B 0,C 180,E1 -2982.786,E2 -2982.786} C_VEL
LIN {X 0,Y 559.945,Z 556.648,A -85,B 0,C 180,E1 -2983.611,E2 -2983.611} C_VEL
LIN {X 0,Y 560.162,Z 544.158,A -85,B 0,C 180,E1 -2984.254,E2 -2984.254} C_VEL
LIN {X 0,Y 560.389,Z 530.444,A -85,B 0,C 180,E1 -2984.798,E2 -2984.798} C_VEL
LIN {X 0,Y 560.553,Z 516.687,A -85,B 0,C 180,E1 -2985.192,E2 -2985.192} C_VEL
LIN {X 0,Y 560.425,Z 509.313,A -85,B 0,C 180,E1 -2985.35,E2 -2985.35} C_VEL
LIN {X 0,Y 559.004,Z 502.186,A -85,B 0,C 180,E1 -2985.519,E2 -2985.519} C_VEL
LIN {X 0,Y 559.108,Z 492.666,A -85,B 0,C 180,E1 -2988.315,E2 -2988.315} C_VEL
LIN {X 0,Y 559.172,Z 483.706,A -85,B 0,C 180,E1 -2990.99,E2 -2990.99} C_VEL
LIN {X 0,Y 559.288,Z 474.747,A -85,B 0,C 180,E1 -2993.71,E2 -2993.71} C_VEL
LIN {X 0,Y 559.441,Z 465.675,A -85,B 0,C 180,E1 -2996.48,E2 -2996.48} C_VEL
LIN {X 0,Y 559.525,Z 456.572,A -85,B 0,C 180,E1 -2999.331,E2 -2999.331} C_VEL
LIN {X 0,Y 559.667,Z 447.45,A -85,B 0,C 180,E1 -3002.255,E2 -3002.255} C_VEL
LIN {X 0,Y 559.81,Z 438.527,A -85,B 0,C 180,E1 -3005.274,E2 -3005.274} C_VEL
LIN {X 0,Y 559.98,Z 431.011,A -85,B 0,C 180,E1 -3007.949,E2 -3007.949} C_VEL
LIN {X 0,Y 559.684,Z 427.285,A -85,B 0,C 180,E1 -3009.354,E2 -3009.354} C_VEL
LIN {X 0,Y 559.183,Z 424.459,A -85,B 0,C 180,E1 -3010.527,E2 -3010.527} C_VEL
LIN {X 0,Y 559.143,Z 424.463,A -85,B 0,C 180,E1 -3013.196,E2 -3013.196} C_VEL
LIN {X 0,Y 559.159,Z 424.462,A -85,B 0,C 180,E1 -3016.268,E2 -3016.268} C_VEL
LIN {X 0,Y 559.173,Z 424.461,A -85,B 0,C 180,E1 -3019.189,E2 -3019.189} C_VEL
LIN {X 0,Y 559.131,Z 424.466,A -85,B 0,C 180,E1 -3021.982,E2 -3021.982} C_VEL
LIN {X 0,Y 559.142,Z 424.464,A -85,B 0,C 180,E1 -3024.784,E2 -3024.784} C_VEL
LIN {X 0,Y 559.17,Z 424.462,A -85,B 0,C 180,E1 -3027.361,E2 -3027.361} C_VEL
LIN {X 0,Y 559.184,Z 424.459,A -85,B 0,C 180,E1 -3030.135,E2 -3030.135} C_VEL
LIN {X 0,Y 559.178,Z 424.458,A -85,B 0,C 180,E1 -3033.169,E2 -3033.169} C_VEL
LIN {X 0,Y 559.151,Z 424.463,A -85,B 0,C 180,E1 -3035.495,E2 -3035.495} C_VEL
LIN {X 0,Y 559.171,Z 424.459,A -85,B 0,C 180,E1 -3038.624,E2 -3038.624} C_VEL
LIN {X 0,Y 559.166,Z 424.46,A -85,B 0,C 180,E1 -3040.926,E2 -3040.926} C_VEL
LIN {X 0,Y 559.167,Z 424.461,A -85,B 0,C 180,E1 -3043.948,E2 -3043.948} C_VEL
LIN {X 0,Y 559.167,Z 424.458,A -85,B 0,C 180,E1 -3046.184,E2 -3046.184} C_VEL
LIN {X 0,Y 559.204,Z 424.455,A -85,B 0,C 180,E1 -3049.134,E2 -3049.134} C_VEL
LIN {X 0,Y 559.205,Z 424.456,A -85,B 0,C 180,E1 -3052.054,E2 -3052.054} C_VEL
LIN {X 0,Y 559.254,Z 424.45,A -85,B 0,C 180,E1 -3054.953,E2 -3054.953} C_VEL
LIN {X 0,Y 559.246,Z 424.45,A -85,B 0,C 180,E1 -3057.84,E2 -3057.84} C_VEL
LIN {X 0,Y 559.269,Z 424.446,A -85,B 0,C 180,E1 -3060.72,E2 -3060.72} C_VEL
LIN {X 0,Y 559.24,Z 424.451,A -85,B 0,C 180,E1 -3062.882,E2 -3062.882} C_VEL
LIN {X 0,Y 559.236,Z 424.452,A -85,B 0,C 180,E1 -3065.77,E2 -3065.77} C_VEL
LIN {X 0,Y 559.197,Z 424.457,A -85,B 0,C 180,E1 -3068.674,E2 -3068.674} C_VEL
LIN {X 0,Y 559.198,Z 424.456,A -85,B 0,C 180,E1 -3071.601,E2 -3071.601} C_VEL
LIN {X 0,Y 559.193,Z 424.455,A -85,B 0,C 180,E1 -3074.596,E2 -3074.596} C_VEL
LIN {X 0,Y 559.158,Z 424.458,A -85,B 0,C 180,E1 -3077.557,E2 -3077.557} C_VEL
LIN {X 0,Y 559.17,Z 424.46,A -85,B 0,C 180,E1 -3079.838,E2 -3079.838} C_VEL
LIN {X 0,Y 559.138,Z 424.464,A -85,B 0,C 180,E1 -3082.153,E2 -3082.153} C_VEL
LIN {X 0,Y 559.174,Z 424.46,A -85,B 0,C 180,E1 -3085.188,E2 -3085.188} C_VEL
LIN {X 0,Y 559.187,Z 424.458,A -85,B 0,C 180,E1 -3087.712,E2 -3087.712} C_VEL
LIN {X 0,Y 559.141,Z 424.459,A -85,B 0,C 180,E1 -3090.629,E2 -3090.629} C_VEL
LIN {X 0,Y 558.483,Z 424.543,A -85,B 0,C 180,E1 -3091.231,E2 -3091.231} C_VEL
LIN {X 0,Y 555.621,Z 424.901,A -85,B 0,C 180,E1 -3092.207,E2 -3092.207} C_VEL
LIN {X 0,Y 553.207,Z 425.201,A -85,B 0,C 180,E1 -3092.993,E2 -3092.993} C_VEL
LIN {X 0,Y 552.185,Z 425.329,A -85,B 0,C 180,E1 -3093.599,E2 -3093.599} C_VEL
LIN {X 0,Y 552.11,Z 425.336,A -85,B 0,C 180,E1 -3093.805,E2 -3093.805} C_VEL
LIN {X 0,Y 552.108,Z 425.337,A -85,B 0,C 180,E1 -3096.747,E2 -3096.747} C_VEL
LIN {X 0,Y 552.127,Z 425.334,A -85,B 0,C 180,E1 -3099.528,E2 -3099.528} C_VEL
LIN {X 0,Y 552.129,Z 425.335,A -85,B 0,C 180,E1 -3102.426,E2 -3102.426} C_VEL
LIN {X 0,Y 552.098,Z 425.34,A -85,B 0,C 180,E1 -3105.564,E2 -3105.564} C_VEL
LIN {X 0,Y 552.131,Z 425.336,A -85,B 0,C 180,E1 -3108.678,E2 -3108.678} C_VEL
LIN {X 0,Y 552.12,Z 425.338,A -85,B 0,C 180,E1 -3111.412,E2 -3111.412} C_VEL
LIN {X 0,Y 552.114,Z 425.338,A -85,B 0,C 180,E1 -3114.159,E2 -3114.159} C_VEL
LIN {X 0,Y 552.124,Z 425.338,A -85,B 0,C 180,E1 -3116.815,E2 -3116.815} C_VEL
LIN {X 0,Y 552.143,Z 425.333,A -85,B 0,C 180,E1 -3119.945,E2 -3119.945} C_VEL
LIN {X 0,Y 552.142,Z 425.332,A -85,B 0,C 180,E1 -3123,E2 -3123} C_VEL
LIN {X 0,Y 552.116,Z 425.338,A -85,B 0,C 180,E1 -3125.162,E2 -3125.162} C_VEL
LIN {X 0,Y 552.129,Z 425.334,A -85,B 0,C 180,E1 -3128.338,E2 -3128.338} C_VEL
LIN {X 0,Y 552.155,Z 425.333,A -85,B 0,C 180,E1 -3130.675,E2 -3130.675} C_VEL
LIN {X 0,Y 552.119,Z 425.336,A -85,B 0,C 180,E1 -3133.738,E2 -3133.738} C_VEL
LIN {X 0,Y 552.14,Z 425.336,A -85,B 0,C 180,E1 -3136.005,E2 -3136.005} C_VEL
LIN {X 0,Y 552.166,Z 425.331,A -85,B 0,C 180,E1 -3138.994,E2 -3138.994} C_VEL
LIN {X 0,Y 552.163,Z 425.33,A -85,B 0,C 180,E1 -3141.952,E2 -3141.952} C_VEL
LIN {X 0,Y 552.23,Z 425.322,A -85,B 0,C 180,E1 -3144.889,E2 -3144.889} C_VEL
LIN {X 0,Y 552.229,Z 425.322,A -85,B 0,C 180,E1 -3147.812,E2 -3147.812} C_VEL
LIN {X 0,Y 552.244,Z 425.32,A -85,B 0,C 180,E1 -3150.729,E2 -3150.729} C_VEL
LIN {X 0,Y 552.208,Z 425.325,A -85,B 0,C 180,E1 -3152.918,E2 -3152.918} C_VEL
LIN {X 0,Y 552.206,Z 425.325,A -85,B 0,C 180,E1 -3155.844,E2 -3155.844} C_VEL
LIN {X 0,Y 552.151,Z 425.332,A -85,B 0,C 180,E1 -3158.786,E2 -3158.786} C_VEL
LIN {X 0,Y 552.167,Z 425.331,A -85,B 0,C 180,E1 -3161.75,E2 -3161.75} C_VEL
LIN {X 0,Y 552.141,Z 425.336,A -85,B 0,C 180,E1 -3164.748,E2 -3164.748} C_VEL
LIN {X 0,Y 552.112,Z 425.338,A -85,B 0,C 180,E1 -3167.788,E2 -3167.788} C_VEL
LIN {X 0,Y 552.13,Z 425.337,A -85,B 0,C 180,E1 -3170.101,E2 -3170.101} C_VEL
LIN {X 0,Y 552.098,Z 425.338,A -85,B 0,C 180,E1 -3172.45,E2 -3172.45} C_VEL
LIN {X 0,Y 552.158,Z 425.332,A -85,B 0,C 180,E1 -3175.35,E2 -3175.35} C_VEL
LIN {X 0,Y 552.128,Z 425.335,A -85,B 0,C 180,E1 -3178.097,E2 -3178.097} C_VEL
LIN {X 0,Y 552.11,Z 425.337,A -85,B 0,C 180,E1 -3180.608,E2 -3180.608} C_VEL
LIN {X 0,Y 552.103,Z 425.338,A -85,B 0,C 180,E1 -3183.186,E2 -3183.186} C_VEL
LIN {X 0,Y 551.904,Z 425.367,A -85,B 0,C 180,E1 -3185.857,E2 -3185.857} C_VEL
LIN {X 0,Y 551.853,Z 426.845,A -85,B 0,C 180,E1 -3187.682,E2 -3187.682} C_VEL
LIN {X 0,Y 551.79,Z 429.668,A -85,B 0,C 180,E1 -3190.509,E2 -3190.509} C_VEL
LIN {X 0,Y 551.818,Z 432.609,A -85,B 0,C 180,E1 -3193.451,E2 -3193.451} C_VEL
LIN {X 0,Y 551.777,Z 435.742,A -85,B 0,C 180,E1 -3196.552,E2 -3196.552} C_VEL
LIN {X 0,Y 551.712,Z 438.674,A -85,B 0,C 180,E1 -3199.483,E2 -3199.483} C_VEL
LIN {X 0,Y 551.692,Z 441.701,A -85,B 0,C 180,E1 -3202.304,E2 -3202.304} C_VEL
LIN {X 0,Y 551.659,Z 444.807,A -85,B 0,C 180,E1 -3205.02,E2 -3205.02} C_VEL
LIN {X 0,Y 551.69,Z 446.39,A -85,B 0,C 180,E1 -3206.39,E2 -3206.39} C_VEL
LIN {X 0,Y 553.658,Z 456.187,A -85,B 0,C 180,E1 -3206.647,E2 -3206.647} C_VEL
LIN {X 0,Y 553.507,Z 470.002,A -85,B 0,C 180,E1 -3207.043,E2 -3207.043} C_VEL
LIN {X 0,Y 553.245,Z 483.825,A -85,B 0,C 180,E1 -3207.594,E2 -3207.594} C_VEL
LIN {X 0,Y 553.018,Z 497.011,A -85,B 0,C 180,E1 -3208.282,E2 -3208.282} C_VEL
LIN {X 0,Y 552.755,Z 509.67,A -85,B 0,C 180,E1 -3209.113,E2 -3209.113} C_VEL
LIN {X 0,Y 552.514,Z 520.633,A -85,B 0,C 180,E1 -3209.995,E2 -3209.995} C_VEL
LIN {X 0,Y 552.313,Z 531.79,A -85,B 0,C 180,E1 -3211.083,E2 -3211.083} C_VEL
LIN {X 0,Y 552.076,Z 540.477,A -85,B 0,C 180,E1 -3212.106,E2 -3212.106} C_VEL
LIN {X 0,Y 551.984,Z 548.805,A -85,B 0,C 180,E1 -3213.282,E2 -3213.282} C_VEL
LIN {X 0,Y 551.867,Z 555.036,A -85,B 0,C 180,E1 -3214.342,E2 -3214.342} C_VEL
LIN {X 0,Y 551.795,Z 560.898,A -85,B 0,C 180,E1 -3215.547,E2 -3215.547} C_VEL
LIN {X 0,Y 551.763,Z 565.568,A -85,B 0,C 180,E1 -3216.743,E2 -3216.743} C_VEL
LIN {X 0,Y 551.71,Z 569.183,A -85,B 0,C 180,E1 -3217.927,E2 -3217.927} C_VEL
LIN {X 0,Y 551.657,Z 571.79,A -85,B 0,C 180,E1 -3219.101,E2 -3219.101} C_VEL
LIN {X 0,Y 551.677,Z 573.903,A -85,B 0,C 180,E1 -3220.657,E2 -3220.657} C_VEL
LIN {X 0,Y 551.651,Z 574.474,A -85,B 0,C 180,E1 -3222.196,E2 -3222.196} C_VEL
LIN {X 0,Y 551.635,Z 573.601,A -85,B 0,C 180,E1 -3223.722,E2 -3223.722} C_VEL
LIN {X 0,Y 551.673,Z 571.294,A -85,B 0,C 180,E1 -3225.239,E2 -3225.239} C_VEL
LIN {X 0,Y 551.724,Z 567.526,A -85,B 0,C 180,E1 -3226.745,E2 -3226.745} C_VEL
LIN {X 0,Y 551.766,Z 563.669,A -85,B 0,C 180,E1 -3227.868,E2 -3227.868} C_VEL
LIN {X 0,Y 551.836,Z 558.901,A -85,B 0,C 180,E1 -3228.987,E2 -3228.987} C_VEL
LIN {X 0,Y 551.946,Z 551.999,A -85,B 0,C 180,E1 -3230.287,E2 -3230.287} C_VEL
LIN {X 0,Y 552.031,Z 543.489,A -85,B 0,C 180,E1 -3231.581,E2 -3231.581} C_VEL
LIN {X 0,Y 552.274,Z 534.614,A -85,B 0,C 180,E1 -3232.689,E2 -3232.689} C_VEL
LIN {X 0,Y 552.451,Z 523.958,A -85,B 0,C 180,E1 -3233.792,E2 -3233.792} C_VEL
LIN {X 0,Y 552.706,Z 512.053,A -85,B 0,C 180,E1 -3234.802,E2 -3234.802} C_VEL
LIN {X 0,Y 552.928,Z 500.101,A -85,B 0,C 180,E1 -3235.626,E2 -3235.626} C_VEL
LIN {X 0,Y 553.213,Z 486.772,A -85,B 0,C 180,E1 -3236.358,E2 -3236.358} C_VEL
LIN {X 0,Y 553.457,Z 473.94,A -85,B 0,C 180,E1 -3236.906,E2 -3236.906} C_VEL
LIN {X 0,Y 553.634,Z 460.251,A -85,B 0,C 180,E1 -3237.34,E2 -3237.34} C_VEL
LIN {X 0,Y 553.446,Z 455.046,A -85,B 0,C 180,E1 -3237.475,E2 -3237.475} C_VEL
LIN {X 0,Y 551.65,Z 446.396,A -85,B 0,C 180,E1 -3237.695,E2 -3237.695} C_VEL
LIN {X 0,Y 551.7,Z 443.737,A -85,B 0,C 180,E1 -3240,E2 -3240} C_VEL
LIN {X 0,Y 551.729,Z 440.419,A -85,B 0,C 180,E1 -3242.92,E2 -3242.92} C_VEL
LIN {X 0,Y 551.768,Z 438.333,A -85,B 0,C 180,E1 -3245.115,E2 -3245.115} C_VEL
LIN {X 0,Y 551.846,Z 436.367,A -85,B 0,C 180,E1 -3247.317,E2 -3247.317} C_VEL
LIN {X 0,Y 551.885,Z 433.756,A -85,B 0,C 180,E1 -3250.27,E2 -3250.27} C_VEL
LIN {X 0,Y 551.898,Z 431.644,A -85,B 0,C 180,E1 -3252.502,E2 -3252.502} C_VEL
LIN {X 0,Y 551.947,Z 429.65,A -85,B 0,C 180,E1 -3254.753,E2 -3254.753} C_VEL
LIN {X 0,Y 551.988,Z 426.819,A -85,B 0,C 180,E1 -3257.792,E2 -3257.792} C_VEL
LIN {X 0,Y 552.022,Z 425.352,A -85,B 0,C 180,E1 -3259.33,E2 -3259.33} C_VEL
LIN {X 0,Y 552.101,Z 425.338,A -85,B 0,C 180,E1 -3261.683,E2 -3261.683} C_VEL
LIN {X 0,Y 552.102,Z 425.342,A -85,B 0,C 180,E1 -3264.038,E2 -3264.038} C_VEL
LIN {X 0,Y 552.129,Z 425.336,A -85,B 0,C 180,E1 -3266.456,E2 -3266.456} C_VEL
LIN {X 0,Y 552.112,Z 425.333,A -85,B 0,C 180,E1 -3268.928,E2 -3268.928} C_VEL
LIN {X 0,Y 552.13,Z 425.333,A -85,B 0,C 180,E1 -3271.48,E2 -3271.48} C_VEL
LIN {X 0,Y 552.141,Z 425.336,A -85,B 0,C 180,E1 -3274.173,E2 -3274.173} C_VEL
LIN {X 0,Y 552.107,Z 425.334,A -85,B 0,C 180,E1 -3276.747,E2 -3276.747} C_VEL
LIN {X 0,Y 552.13,Z 425.335,A -85,B 0,C 180,E1 -3279.527,E2 -3279.527} C_VEL
LIN {X 0,Y 552.127,Z 425.335,A -85,B 0,C 180,E1 -3282.426,E2 -3282.426} C_VEL
LIN {X 0,Y 552.096,Z 425.343,A -85,B 0,C 180,E1 -3285.563,E2 -3285.563} C_VEL
LIN {X 0,Y 552.137,Z 425.336,A -85,B 0,C 180,E1 -3288.677,E2 -3288.677} C_VEL
LIN {X 0,Y 552.205,Z 425.657,A -85,B 0,C 180,E1 -3289.047,E2 -3289.047} C_VEL
LIN {X 0,Y 552.849,Z 429.513,A -85,B 0,C 180,E1 -3290.846,E2 -3290.846} C_VEL
LIN {X 0,Y 552.923,Z 434.376,A -85,B 0,C 180,E1 -3292.851,E2 -3292.851} C_VEL
LIN {X 0,Y 552.677,Z 442.193,A -85,B 0,C 180,E1 -3295.747,E2 -3295.747} C_VEL
LIN {X 0,Y 552.544,Z 450.428,A -85,B 0,C 180,E1 -3298.568,E2 -3298.568} C_VEL
LIN {X 0,Y 552.404,Z 459.382,A -85,B 0,C 180,E1 -3301.385,E2 -3301.385} C_VEL
LIN {X 0,Y 552.304,Z 467.767,A -85,B 0,C 180,E1 -3303.96,E2 -3303.96} C_VEL
LIN {X 0,Y 552.239,Z 477.228,A -85,B 0,C 180,E1 -3306.765,E2 -3306.765} C_VEL
LIN {X 0,Y 552.103,Z 486.266,A -85,B 0,C 180,E1 -3309.509,E2 -3309.509} C_VEL
LIN {X 0,Y 552.028,Z 495.226,A -85,B 0,C 180,E1 -3312.209,E2 -3312.209} C_VEL
LIN {X 0,Y 551.968,Z 502.186,A -85,B 0,C 180,E1 -3314.279,E2 -3314.279} C_VEL
LIN {X 0,Y 553.733,Z 512.18,A -85,B 0,C 180,E1 -3314.519,E2 -3314.519} C_VEL
LIN {X 0,Y 553.54,Z 526.594,A -85,B 0,C 180,E1 -3314.888,E2 -3314.888} C_VEL
LIN {X 0,Y 553.307,Z 539.971,A -85,B 0,C 180,E1 -3315.378,E2 -3315.378} C_VEL
LIN {X 0,Y 553.123,Z 553.4,A -85,B 0,C 180,E1 -3316.03,E2 -3316.03} C_VEL
LIN {X 0,Y 552.838,Z 565.518,A -85,B 0,C 180,E1 -3316.772,E2 -3316.772} C_VEL
LIN {X 0,Y 552.594,Z 577.753,A -85,B 0,C 180,E1 -3317.7,E2 -3317.7} C_VEL
LIN {X 0,Y 552.399,Z 589.057,A -85,B 0,C 180,E1 -3318.754,E2 -3318.754} C_VEL
LIN {X 0,Y 552.121,Z 599.34,A -85,B 0,C 180,E1 -3319.92,E2 -3319.92} C_VEL
LIN {X 0,Y 552.008,Z 607.408,A -85,B 0,C 180,E1 -3321.027,E2 -3321.027} C_VEL
LIN {X 0,Y 551.9,Z 615.136,A -85,B 0,C 180,E1 -3322.316,E2 -3322.316} C_VEL
LIN {X 0,Y 551.784,Z 621.636,A -85,B 0,C 180,E1 -3323.67,E2 -3323.67} C_VEL
LIN {X 0,Y 551.716,Z 626.201,A -85,B 0,C 180,E1 -3324.884,E2 -3324.884} C_VEL
LIN {X 0,Y 551.74,Z 630.316,A -85,B 0,C 180,E1 -3326.348,E2 -3326.348} C_VEL
LIN {X 0,Y 551.655,Z 633.001,A -85,B 0,C 180,E1 -3327.81,E2 -3327.81} C_VEL
LIN {X 0,Y 551.639,Z 634.333,A -85,B 0,C 180,E1 -3329.27,E2 -3329.27} C_VEL
LIN {X 0,Y 551.639,Z 634.333,A -85,B 0,C 180,E1 -3330.73,E2 -3330.73} C_VEL
LIN {X 0,Y 551.655,Z 633.003,A -85,B 0,C 180,E1 -3332.19,E2 -3332.19} C_VEL
LIN {X 0,Y 551.74,Z 630.319,A -85,B 0,C 180,E1 -3333.652,E2 -3333.652} C_VEL
LIN {X 0,Y 551.716,Z 626.202,A -85,B 0,C 180,E1 -3335.116,E2 -3335.116} C_VEL
LIN {X 0,Y 551.786,Z 621.626,A -85,B 0,C 180,E1 -3336.332,E2 -3336.332} C_VEL
LIN {X 0,Y 551.9,Z 615.136,A -85,B 0,C 180,E1 -3337.684,E2 -3337.684} C_VEL
LIN {X 0,Y 552.01,Z 607.408,A -85,B 0,C 180,E1 -3338.972,E2 -3338.972} C_VEL
LIN {X 0,Y 552.121,Z 599.339,A -85,B 0,C 180,E1 -3340.08,E2 -3340.08} C_VEL
LIN {X 0,Y 552.401,Z 589.092,A -85,B 0,C 180,E1 -3341.242,E2 -3341.242} C_VEL
LIN {X 0,Y 552.594,Z 577.752,A -85,B 0,C 180,E1 -3342.3,E2 -3342.3} C_VEL
LIN {X 0,Y 552.838,Z 565.52,A -85,B 0,C 180,E1 -3343.228,E2 -3343.228} C_VEL
LIN {X 0,Y 553.123,Z 553.402,A -85,B 0,C 180,E1 -3343.97,E2 -3343.97} C_VEL
LIN {X 0,Y 553.322,Z 539.964,A -85,B 0,C 180,E1 -3344.622,E2 -3344.622} C_VEL
LIN {X 0,Y 553.525,Z 525.577,A -85,B 0,C 180,E1 -3345.144,E2 -3345.144} C_VEL
LIN {X 0,Y 553.733,Z 511.035,A -85,B 0,C 180,E1 -3345.505,E2 -3345.505} C_VEL
LIN {X 0,Y 551.968,Z 502.186,A -85,B 0,C 180,E1 -3345.721,E2 -3345.721} C_VEL
LIN {X 0,Y 552.071,Z 492.666,A -85,B 0,C 180,E1 -3348.557,E2 -3348.557} C_VEL
LIN {X 0,Y 552.155,Z 483.706,A -85,B 0,C 180,E1 -3351.269,E2 -3351.269} C_VEL
LIN {X 0,Y 552.267,Z 474.579,A -85,B 0,C 180,E1 -3354.03,E2 -3354.03} C_VEL
LIN {X 0,Y 552.387,Z 466.768,A -85,B 0,C 180,E1 -3356.442,E2 -3356.442} C_VEL
LIN {X 0,Y 552.496,Z 457.682,A -85,B 0,C 180,E1 -3359.323,E2 -3359.323} C_VEL
LIN {X 0,Y 552.667,Z 448.604,A -85,B 0,C 180,E1 -3362.282,E2 -3362.282} C_VEL
LIN {X 0,Y 552.829,Z 440.971,A -85,B 0,C 180,E1 -3364.894,E2 -3364.894} C_VEL
LIN {X 0,Y 553.004,Z 433.476,A -85,B 0,C 180,E1 -3367.59,E2 -3367.59} C_VEL
LIN {X 0,Y 552.839,Z 429.32,A -85,B 0,C 180,E1 -3369.153,E2 -3369.153} C_VEL
LIN {X 0,Y 552.132,Z 425.338,A -85,B 0,C 180,E1 -3370.779,E2 -3370.779} C_VEL
LIN {X 0,Y 552.099,Z 425.342,A -85,B 0,C 180,E1 -3373.482,E2 -3373.482} C_VEL
LIN {X 0,Y 552.116,Z 425.338,A -85,B 0,C 180,E1 -3376.577,E2 -3376.577} C_VEL
LIN {X 0,Y 552.118,Z 425.336,A -85,B 0,C 180,E1 -3379.52,E2 -3379.52} C_VEL
LIN {X 0,Y 552.09,Z 425.34,A -85,B 0,C 180,E1 -3382.336,E2 -3382.336} C_VEL
LIN {X 0,Y 552.116,Z 425.337,A -85,B 0,C 180,E1 -3385.053,E2 -3385.053} C_VEL
LIN {X 0,Y 552.124,Z 425.336,A -85,B 0,C 180,E1 -3387.682,E2 -3387.682} C_VEL
LIN {X 0,Y 552.14,Z 425.337,A -85,B 0,C 180,E1 -3390.237,E2 -3390.237} C_VEL
LIN {X 0,Y 552.143,Z 425.336,A -85,B 0,C 180,E1 -3392.997,E2 -3392.997} C_VEL
LIN {X 0,Y 552.107,Z 425.338,A -85,B 0,C 180,E1 -3395.161,E2 -3395.161} C_VEL
LIN {X 0,Y 552.091,Z 425.339,A -85,B 0,C 180,E1 -3397.549,E2 -3397.549} C_VEL
LIN {X 0,Y 552.143,Z 425.333,A -85,B 0,C 180,E1 -3400.373,E2 -3400.373} C_VEL
LIN {X 0,Y 552.152,Z 425.332,A -85,B 0,C 180,E1 -3402.977,E2 -3402.977} C_VEL
LIN {X 0,Y 552.13,Z 425.334,A -85,B 0,C 180,E1 -3406.004,E2 -3406.004} C_VEL
LIN {X 0,Y 552.172,Z 425.33,A -85,B 0,C 180,E1 -3408.994,E2 -3408.994} C_VEL
LIN {X 0,Y 552.158,Z 425.333,A -85,B 0,C 180,E1 -3411.952,E2 -3411.952} C_VEL
LIN {X 0,Y 552.228,Z 425.326,A -85,B 0,C 180,E1 -3414.889,E2 -3414.889} C_VEL
LIN {X 0,Y 552.218,Z 425.326,A -85,B 0,C 180,E1 -3417.812,E2 -3417.812} C_VEL
LIN {X 0,Y 552.239,Z 425.322,A -85,B 0,C 180,E1 -3420.729,E2 -3420.729} C_VEL
LIN {X 0,Y 552.206,Z 425.328,A -85,B 0,C 180,E1 -3422.918,E2 -3422.918} C_VEL
LIN {X 0,Y 552.206,Z 425.328,A -85,B 0,C 180,E1 -3425.844,E2 -3425.844} C_VEL
LIN {X 0,Y 552.165,Z 425.332,A -85,B 0,C 180,E1 -3428.786,E2 -3428.786} C_VEL
LIN {X 0,Y 552.156,Z 425.332,A -85,B 0,C 180,E1 -3431.751,E2 -3431.751} C_VEL
LIN {X 0,Y 552.13,Z 425.334,A -85,B 0,C 180,E1 -3434.749,E2 -3434.749} C_VEL
LIN {X 0,Y 552.109,Z 425.337,A -85,B 0,C 180,E1 -3437.789,E2 -3437.789} C_VEL
LIN {X 0,Y 552.129,Z 425.335,A -85,B 0,C 180,E1 -3440.101,E2 -3440.101} C_VEL
LIN {X 0,Y 552.091,Z 425.342,A -85,B 0,C 180,E1 -3442.451,E2 -3442.451} C_VEL
LIN {X 0,Y 552.15,Z 425.334,A -85,B 0,C 180,E1 -3445.351,E2 -3445.351} C_VEL
LIN {X 0,Y 552.121,Z 425.337,A -85,B 0,C 180,E1 -3448.098,E2 -3448.098} C_VEL
LIN {X 0,Y 552.102,Z 425.341,A -85,B 0,C 180,E1 -3450.625,E2 -3450.625} C_VEL
LIN {X 0,Y 552.119,Z 425.339,A -85,B 0,C 180,E1 -3453.186,E2 -3453.186} C_VEL
LIN {X 0,Y 552.11,Z 425.336,A -85,B 0,C 180,E1 -3453.805,E2 -3453.805} C_VEL
LIN {X 0,Y 551.474,Z 425.419,A -85,B 0,C 180,E1 -3454.413,E2 -3454.413} C_VEL
LIN {X 0,Y 548.652,Z 425.767,A -85,B 0,C 180,E1 -3455.402,E2 -3455.402} C_VEL
LIN {X 0,Y 546.231,Z 426.072,A -85,B 0,C 180,E1 -3456.197,E2 -3456.197} C_VEL
LIN {X 0,Y 545.162,Z 426.202,A -85,B 0,C 180,E1 -3456.811,E2 -3456.811} C_VEL
LIN {X 0,Y 545.061,Z 426.215,A -85,B 0,C 180,E1 -3457.019,E2 -3457.019} C_VEL
LIN {X 0,Y 545.063,Z 426.218,A -85,B 0,C 180,E1 -3460.143,E2 -3460.143} C_VEL
LIN {X 0,Y 545.086,Z 426.215,A -85,B 0,C 180,E1 -3463.106,E2 -3463.106} C_VEL
LIN {X 0,Y 545.066,Z 426.215,A -85,B 0,C 180,E1 -3466.225,E2 -3466.225} C_VEL
LIN {X 0,Y 545.09,Z 426.211,A -85,B 0,C 180,E1 -3468.887,E2 -3468.887} C_VEL
LIN {X 0,Y 545.054,Z 426.216,A -85,B 0,C 180,E1 -3471.764,E2 -3471.764} C_VEL
LIN {X 0,Y 545.066,Z 426.214,A -85,B 0,C 180,E1 -3474.535,E2 -3474.535} C_VEL
LIN {X 0,Y 545.082,Z 426.212,A -85,B 0,C 180,E1 -3477.213,E2 -3477.213} C_VEL
LIN {X 0,Y 545.104,Z 426.211,A -85,B 0,C 180,E1 -3479.814,E2 -3479.814} C_VEL
LIN {X 0,Y 545.095,Z 426.21,A -85,B 0,C 180,E1 -3482.827,E2 -3482.827} C_VEL
LIN {X 0,Y 545.052,Z 426.216,A -85,B 0,C 180,E1 -3485.631,E2 -3485.631} C_VEL
LIN {X 0,Y 545.069,Z 426.216,A -85,B 0,C 180,E1 -3488.837,E2 -3488.837} C_VEL
LIN {X 0,Y 545.079,Z 426.213,A -85,B 0,C 180,E1 -3491.196,E2 -3491.196} C_VEL
LIN {X 0,Y 545.076,Z 426.214,A -85,B 0,C 180,E1 -3493.522,E2 -3493.522} C_VEL
LIN {X 0,Y 545.099,Z 426.214,A -85,B 0,C 180,E1 -3495.82,E2 -3495.82} C_VEL
LIN {X 0,Y 545.122,Z 426.21,A -85,B 0,C 180,E1 -3498.85,E2 -3498.85} C_VEL
LIN {X 0,Y 545.133,Z 426.206,A -85,B 0,C 180,E1 -3501.847,E2 -3501.847} C_VEL
LIN {X 0,Y 545.205,Z 426.197,A -85,B 0,C 180,E1 -3504.823,E2 -3504.823} C_VEL
LIN {X 0,Y 545.201,Z 426.198,A -85,B 0,C 180,E1 -3507.784,E2 -3507.784} C_VEL
LIN {X 0,Y 545.214,Z 426.196,A -85,B 0,C 180,E1 -3510.739,E2 -3510.739} C_VEL
LIN {X 0,Y 545.175,Z 426.201,A -85,B 0,C 180,E1 -3512.956,E2 -3512.956} C_VEL
LIN {X 0,Y 545.178,Z 426.2,A -85,B 0,C 180,E1 -3515.919,E2 -3515.919} C_VEL
LIN {X 0,Y 545.113,Z 426.209,A -85,B 0,C 180,E1 -3518.9,E2 -3518.9} C_VEL
LIN {X 0,Y 545.139,Z 426.208,A -85,B 0,C 180,E1 -3521.904,E2 -3521.904} C_VEL
LIN {X 0,Y 545.089,Z 426.214,A -85,B 0,C 180,E1 -3524.943,E2 -3524.943} C_VEL
LIN {X 0,Y 545.08,Z 426.212,A -85,B 0,C 180,E1 -3528.025,E2 -3528.025} C_VEL
LIN {X 0,Y 545.095,Z 426.214,A -85,B 0,C 180,E1 -3530.372,E2 -3530.372} C_VEL
LIN {X 0,Y 545.095,Z 426.211,A -85,B 0,C 180,E1 -3533.558,E2 -3533.558} C_VEL
LIN {X 0,Y 545.082,Z 426.214,A -85,B 0,C 180,E1 -3536,E2 -3536} C_VEL
LIN {X 0,Y 545.093,Z 426.213,A -85,B 0,C 180,E1 -3538.748,E2 -3538.748} C_VEL
LIN {X 0,Y 545.077,Z 426.213,A -85,B 0,C 180,E1 -3541.681,E2 -3541.681} C_VEL
LIN {X 0,Y 544.996,Z 426.227,A -85,B 0,C 180,E1 -3544.379,E2 -3544.379} C_VEL
LIN {X 0,Y 544.792,Z 426.253,A -85,B 0,C 180,E1 -3546.399,E2 -3546.399} C_VEL
LIN {X 0,Y 544.748,Z 429.068,A -85,B 0,C 180,E1 -3549.278,E2 -3549.278} C_VEL
LIN {X 0,Y 544.712,Z 431.891,A -85,B 0,C 180,E1 -3552.137,E2 -3552.137} C_VEL
LIN {X 0,Y 544.682,Z 434.545,A -85,B 0,C 180,E1 -3554.792,E2 -3554.792} C_VEL
LIN {X 0,Y 544.68,Z 437.09,A -85,B 0,C 180,E1 -3557.346,E2 -3557.346} C_VEL
LIN {X 0,Y 544.631,Z 439.54,A -85,B 0,C 180,E1 -3559.818,E2 -3559.818} C_VEL
LIN {X 0,Y 544.573,Z 442.416,A -85,B 0,C 180,E1 -3562.658,E2 -3562.658} C_VEL
LIN {X 0,Y 544.598,Z 446.011,A -85,B 0,C 180,E1 -3565.85,E2 -3565.85} C_VEL
LIN {X 0,Y 544.601,Z 446.383,A -85,B 0,C 180,E1 -3566.176,E2 -3566.176} C_VEL
LIN {X 0,Y 546.805,Z 457.388,A -85,B 0,C 180,E1 -3566.48,E2 -3566.48} C_VEL
LIN {X 0,Y 546.619,Z 471.457,A -85,B 0,C 180,E1 -3566.903,E2 -3566.903} C_VEL
LIN {X 0,Y 546.363,Z 485.319,A -85,B 0,C 180,E1 -3567.479,E2 -3567.479} C_VEL
LIN {X 0,Y 546.09,Z 497.825,A -85,B 0,C 180,E1 -3568.152,E2 -3568.152} C_VEL
LIN {X 0,Y 545.797,Z 510.391,A -85,B 0,C 180,E1 -3568.998,E2 -3568.998} C_VEL
LIN {X 0,Y 545.498,Z 521.824,A -85,B 0,C 180,E1 -3569.943,E2 -3569.943} C_VEL
LIN {X 0,Y 545.303,Z 532.208,A -85,B 0,C 180,E1 -3570.986,E2 -3570.986} C_VEL
LIN {X 0,Y 545.022,Z 541.653,A -85,B 0,C 180,E1 -3572.131,E2 -3572.131} C_VEL
LIN {X 0,Y 544.895,Z 550.061,A -85,B 0,C 180,E1 -3573.371,E2 -3573.371} C_VEL
LIN {X 0,Y 544.801,Z 556.67,A -85,B 0,C 180,E1 -3574.554,E2 -3574.554} C_VEL
LIN {X 0,Y 544.704,Z 563.182,A -85,B 0,C 180,E1 -3576.02,E2 -3576.02} C_VEL
LIN {X 0,Y 544.636,Z 567.355,A -85,B 0,C 180,E1 -3577.224,E2 -3577.224} C_VEL
LIN {X 0,Y 544.644,Z 570.183,A -85,B 0,C 180,E1 -3578.289,E2 -3578.289} C_VEL
LIN {X 0,Y 544.539,Z 572.674,A -85,B 0,C 180,E1 -3579.606,E2 -3579.606} C_VEL
LIN {X 0,Y 544.576,Z 573.664,A -85,B 0,C 180,E1 -3580.404,E2 -3580.404} C_VEL
LIN {X 0,Y 544.545,Z 574.487,A -85,B 0,C 180,E1 -3581.956,E2 -3581.956} C_VEL
LIN {X 0,Y 544.554,Z 573.854,A -85,B 0,C 180,E1 -3583.505,E2 -3583.505} C_VEL
LIN {X 0,Y 544.553,Z 571.76,A -85,B 0,C 180,E1 -3585.041,E2 -3585.041} C_VEL
LIN {X 0,Y 544.645,Z 568.204,A -85,B 0,C 180,E1 -3586.569,E2 -3586.569} C_VEL
LIN {X 0,Y 544.701,Z 563.123,A -85,B 0,C 180,E1 -3588.086,E2 -3588.086} C_VEL
LIN {X 0,Y 544.752,Z 558.217,A -85,B 0,C 180,E1 -3589.218,E2 -3589.218} C_VEL
LIN {X 0,Y 544.876,Z 551.164,A -85,B 0,C 180,E1 -3590.534,E2 -3590.534} C_VEL
LIN {X 0,Y 545.063,Z 542.464,A -85,B 0,C 180,E1 -3591.846,E2 -3591.846} C_VEL
LIN {X 0,Y 545.292,Z 532.988,A -85,B 0,C 180,E1 -3593.015,E2 -3593.015} C_VEL
LIN {X 0,Y 545.5,Z 522.509,A -85,B 0,C 180,E1 -3594.084,E2 -3594.084} C_VEL
LIN {X 0,Y 545.735,Z 511.473,A -85,B 0,C 180,E1 -3595.013,E2 -3595.013} C_VEL
LIN {X 0,Y 546.05,Z 499.322,A -85,B 0,C 180,E1 -3595.848,E2 -3595.848} C_VEL
LIN {X 0,Y 546.302,Z 487.735,A -85,B 0,C 180,E1 -3596.496,E2 -3596.496} C_VEL
LIN {X 0,Y 546.586,Z 475.177,A -85,B 0,C 180,E1 -3597.052,E2 -3597.052} C_VEL
LIN {X 0,Y 546.792,Z 461.099,A -85,B 0,C 180,E1 -3597.514,E2 -3597.514} C_VEL
LIN {X 0,Y 546.579,Z 456.07,A -85,B 0,C 180,E1 -3597.651,E2 -3597.651} C_VEL
LIN {X 0,Y 544.557,Z 446.379,A -85,B 0,C 180,E1 -3597.92,E2 -3597.92} C_VEL
LIN {X 0,Y 544.599,Z 443.177,A -85,B 0,C 180,E1 -3600.739,E2 -3600.739} C_VEL
LIN {X 0,Y 544.719,Z 440.309,A -85,B 0,C 180,E1 -3603.699,E2 -3603.699} C_VEL
LIN {X 0,Y 544.788,Z 437.646,A -85,B 0,C 180,E1 -3606.667,E2 -3606.667} C_VEL
LIN {X 0,Y 544.789,Z 435.739,A -85,B 0,C 180,E1 -3608.905,E2 -3608.905} C_VEL
LIN {X 0,Y 544.899,Z 433.386,A -85,B 0,C 180,E1 -3611.416,E2 -3611.416} C_VEL
LIN {X 0,Y 544.897,Z 430.438,A -85,B 0,C 180,E1 -3614.688,E2 -3614.688} C_VEL
LIN {X 0,Y 544.954,Z 428.018,A -85,B 0,C 180,E1 -3617.384,E2 -3617.384} C_VEL
LIN {X 0,Y 544.996,Z 426.227,A -85,B 0,C 180,E1 -3619.59,E2 -3619.59} C_VEL
LIN {X 0,Y 545.042,Z 426.221,A -85,B 0,C 180,E1 -3621.959,E2 -3621.959} C_VEL
LIN {X 0,Y 545.047,Z 426.22,A -85,B 0,C 180,E1 -3624.369,E2 -3624.369} C_VEL
LIN {X 0,Y 545.096,Z 426.207,A -85,B 0,C 180,E1 -3627.176,E2 -3627.176} C_VEL
LIN {X 0,Y 545.091,Z 426.214,A -85,B 0,C 180,E1 -3630.25,E2 -3630.25} C_VEL
LIN {X 0,Y 545.087,Z 426.208,A -85,B 0,C 180,E1 -3633.065,E2 -3633.065} C_VEL
LIN {X 0,Y 545.058,Z 426.216,A -85,B 0,C 180,E1 -3635.678,E2 -3635.678} C_VEL
LIN {X 0,Y 545.05,Z 426.219,A -85,B 0,C 180,E1 -3638.237,E2 -3638.237} C_VEL
LIN {X 0,Y 545.097,Z 426.208,A -85,B 0,C 180,E1 -3641.113,E2 -3641.113} C_VEL
LIN {X 0,Y 545.055,Z 426.22,A -85,B 0,C 180,E1 -3644.129,E2 -3644.129} C_VEL
LIN {X 0,Y 545.083,Z 426.214,A -85,B 0,C 180,E1 -3646.895,E2 -3646.895} C_VEL
LIN {X 0,Y 545.107,Z 426.282,A -85,B 0,C 180,E1 -3648.567,E2 -3648.567} C_VEL
LIN {X 0,Y 545.916,Z 431.101,A -85,B 0,C 180,E1 -3650.891,E2 -3650.891} C_VEL
LIN {X 0,Y 545.962,Z 435.575,A -85,B 0,C 180,E1 -3652.771,E2 -3652.771} C_VEL
LIN {X 0,Y 545.714,Z 442.836,A -85,B 0,C 180,E1 -3655.51,E2 -3655.51} C_VEL
LIN {X 0,Y 545.539,Z 451.725,A -85,B 0,C 180,E1 -3658.614,E2 -3658.614} C_VEL
LIN {X 0,Y 545.357,Z 460.721,A -85,B 0,C 180,E1 -3661.523,E2 -3661.523} C_VEL
LIN {X 0,Y 545.245,Z 468.719,A -85,B 0,C 180,E1 -3664.008,E2 -3664.008} C_VEL
LIN {X 0,Y 545.163,Z 478.146,A -85,B 0,C 180,E1 -3666.847,E2 -3666.847} C_VEL
LIN {X 0,Y 545.058,Z 487.546,A -85,B 0,C 180,E1 -3669.627,E2 -3669.627} C_VEL
LIN {X 0,Y 544.974,Z 496.464,A -85,B 0,C 180,E1 -3672.346,E2 -3672.346} C_VEL
LIN {X 0,Y 544.896,Z 502.186,A -85,B 0,C 180,E1 -3674.069,E2 -3674.069} C_VEL
LIN {X 0,Y 546.895,Z 513.32,A -85,B 0,C 180,E1 -3674.344,E2 -3674.344} C_VEL
LIN {X 0,Y 546.685,Z 527.243,A -85,B 0,C 180,E1 -3674.714,E2 -3674.714} C_VEL
LIN {X 0,Y 546.422,Z 541.095,A -85,B 0,C 180,E1 -3675.237,E2 -3675.237} C_VEL
LIN {X 0,Y 546.232,Z 553.402,A -85,B 0,C 180,E1 -3675.85,E2 -3675.85} C_VEL
LIN {X 0,Y 545.918,Z 565.519,A -85,B 0,C 180,E1 -3676.601,E2 -3676.601} C_VEL
LIN {X 0,Y 545.627,Z 577.751,A -85,B 0,C 180,E1 -3677.541,E2 -3677.541} C_VEL
LIN {X 0,Y 545.431,Z 587.846,A -85,B 0,C 180,E1 -3678.481,E2 -3678.481} C_VEL
LIN {X 0,Y 545.175,Z 597.854,A -85,B 0,C 180,E1 -3679.603,E2 -3679.603} C_VEL
LIN {X 0,Y 545,Z 606.175,A -85,B 0,C 180,E1 -3680.724,E2 -3680.724} C_VEL
LIN {X 0,Y 544.833,Z 614.128,A -85,B 0,C 180,E1 -3682.029,E2 -3682.029} C_VEL
LIN {X 0,Y 544.753,Z 620.876,A -85,B 0,C 180,E1 -3683.413,E2 -3683.413} C_VEL
LIN {X 0,Y 544.646,Z 626.201,A -85,B 0,C 180,E1 -3684.818,E2 -3684.818} C_VEL
LIN {X 0,Y 544.657,Z 630.316,A -85,B 0,C 180,E1 -3686.301,E2 -3686.301} C_VEL
LIN {X 0,Y 544.569,Z 633.002,A -85,B 0,C 180,E1 -3687.781,E2 -3687.781} C_VEL
LIN {X 0,Y 544.539,Z 634.333,A -85,B 0,C 180,E1 -3689.261,E2 -3689.261} C_VEL
LIN {X 0,Y 544.539,Z 634.334,A -85,B 0,C 180,E1 -3690.739,E2 -3690.739} C_VEL
LIN {X 0,Y 544.569,Z 633.004,A -85,B 0,C 180,E1 -3692.219,E2 -3692.219} C_VEL
LIN {X 0,Y 544.657,Z 630.319,A -85,B 0,C 180,E1 -3693.699,E2 -3693.699} C_VEL
LIN {X 0,Y 544.646,Z 626.202,A -85,B 0,C 180,E1 -3695.182,E2 -3695.182} C_VEL
LIN {X 0,Y 544.734,Z 620.949,A -85,B 0,C 180,E1 -3696.57,E2 -3696.57} C_VEL
LIN {X 0,Y 544.833,Z 614.129,A -85,B 0,C 180,E1 -3697.971,E2 -3697.971} C_VEL
LIN {X 0,Y 544.999,Z 606.175,A -85,B 0,C 180,E1 -3699.276,E2 -3699.276} C_VEL
LIN {X 0,Y 545.175,Z 597.854,A -85,B 0,C 180,E1 -3700.397,E2 -3700.397} C_VEL
LIN {X 0,Y 545.364,Z 588.03,A -85,B 0,C 180,E1 -3701.501,E2 -3701.501} C_VEL
LIN {X 0,Y 545.667,Z 576.647,A -85,B 0,C 180,E1 -3702.553,E2 -3702.553} C_VEL
LIN {X 0,Y 545.913,Z 564.107,A -85,B 0,C 180,E1 -3703.493,E2 -3703.493} C_VEL
LIN {X 0,Y 546.277,Z 551.646,A -85,B 0,C 180,E1 -3704.244,E2 -3704.244} C_VEL
LIN {X 0,Y 546.499,Z 537.704,A -85,B 0,C 180,E1 -3704.904,E2 -3704.904} C_VEL
LIN {X 0,Y 546.723,Z 523.651,A -85,B 0,C 180,E1 -3705.397,E2 -3705.397} C_VEL
LIN {X 0,Y 546.785,Z 511.676,A -85,B 0,C 180,E1 -3705.694,E2 -3705.694} C_VEL
LIN {X 0,Y 544.895,Z 502.186,A -85,B 0,C 180,E1 -3705.931,E2 -3705.931} C_VEL
LIN {X 0,Y 545.01,Z 492.666,A -85,B 0,C 180,E1 -3708.807,E2 -3708.807} C_VEL
LIN {X 0,Y 545.157,Z 482.303,A -85,B 0,C 180,E1 -3711.953,E2 -3711.953} C_VEL
LIN {X 0,Y 545.255,Z 473.051,A -85,B 0,C 180,E1 -3714.765,E2 -3714.765} C_VEL
LIN {X 0,Y 545.41,Z 463.987,A -85,B 0,C 180,E1 -3717.638,E2 -3717.638} C_VEL
LIN {X 0,Y 545.544,Z 454.777,A -85,B 0,C 180,E1 -3720.634,E2 -3720.634} C_VEL
LIN {X 0,Y 545.728,Z 447.301,A -85,B 0,C 180,E1 -3723.167,E2 -3723.167} C_VEL
LIN {X 0,Y 545.944,Z 439.806,A -85,B 0,C 180,E1 -3725.806,E2 -3725.806} C_VEL
LIN {X 0,Y 546.069,Z 433.104,A -85,B 0,C 180,E1 -3728.272,E2 -3728.272} C_VEL
LIN {X 0,Y 545.504,Z 428.468,A -85,B 0,C 180,E1 -3730.103,E2 -3730.103} C_VEL
LIN {X 0,Y 545.111,Z 426.212,A -85,B 0,C 180,E1 -3731.111,E2 -3731.111} C_VEL
LIN {X 0,Y 545.051,Z 426.218,A -85,B 0,C 180,E1 -3734.129,E2 -3734.129} C_VEL
LIN {X 0,Y 545.083,Z 426.212,A -85,B 0,C 180,E1 -3736.894,E2 -3736.894} C_VEL
LIN {X 0,Y 545.07,Z 426.213,A -85,B 0,C 180,E1 -3739.858,E2 -3739.858} C_VEL
LIN {X 0,Y 545.069,Z 426.216,A -85,B 0,C 180,E1 -3743.073,E2 -3743.073} C_VEL
LIN {X 0,Y 545.071,Z 426.215,A -85,B 0,C 180,E1 -3746.329,E2 -3746.329} C_VEL
LIN {X 0,Y 545.065,Z 426.217,A -85,B 0,C 180,E1 -3748.952,E2 -3748.952} C_VEL
LIN {X 0,Y 545.1,Z 426.213,A -85,B 0,C 180,E1 -3751.508,E2 -3751.508} C_VEL
LIN {X 0,Y 545.094,Z 426.213,A -85,B 0,C 180,E1 -3754.489,E2 -3754.489} C_VEL
LIN {X 0,Y 545.039,Z 426.219,A -85,B 0,C 180,E1 -3757.242,E2 -3757.242} C_VEL
LIN {X 0,Y 545.115,Z 426.208,A -85,B 0,C 180,E1 -3760.415,E2 -3760.415} C_VEL
LIN {X 0,Y 545.072,Z 426.215,A -85,B 0,C 180,E1 -3763.521,E2 -3763.521} C_VEL
LIN {X 0,Y 545.088,Z 426.211,A -85,B 0,C 180,E1 -3765.82,E2 -3765.82} C_VEL
LIN {X 0,Y 545.126,Z 426.207,A -85,B 0,C 180,E1 -3768.85,E2 -3768.85} C_VEL
LIN {X 0,Y 545.128,Z 426.208,A -85,B 0,C 180,E1 -3771.847,E2 -3771.847} C_VEL
LIN {X 0,Y 545.203,Z 426.201,A -85,B 0,C 180,E1 -3774.823,E2 -3774.823} C_VEL
LIN {X 0,Y 545.189,Z 426.202,A -85,B 0,C 180,E1 -3777.784,E2 -3777.784} C_VEL
LIN {X 0,Y 545.209,Z 426.197,A -85,B 0,C 180,E1 -3780.739,E2 -3780.739} C_VEL
LIN {X 0,Y 545.172,Z 426.204,A -85,B 0,C 180,E1 -3782.956,E2 -3782.956} C_VEL
LIN {X 0,Y 545.177,Z 426.204,A -85,B 0,C 180,E1 -3785.92,E2 -3785.92} C_VEL
LIN {X 0,Y 545.122,Z 426.208,A -85,B 0,C 180,E1 -3788.9,E2 -3788.9} C_VEL
LIN {X 0,Y 545.129,Z 426.207,A -85,B 0,C 180,E1 -3791.905,E2 -3791.905} C_VEL
LIN {X 0,Y 545.079,Z 426.213,A -85,B 0,C 180,E1 -3794.944,E2 -3794.944} C_VEL
LIN {X 0,Y 545.077,Z 426.215,A -85,B 0,C 180,E1 -3798.026,E2 -3798.026} C_VEL
LIN {X 0,Y 545.094,Z 426.211,A -85,B 0,C 180,E1 -3800.372,E2 -3800.372} C_VEL
LIN {X 0,Y 545.087,Z 426.214,A -85,B 0,C 180,E1 -3803.559,E2 -3803.559} C_VEL
LIN {X 0,Y 545.075,Z 426.214,A -85,B 0,C 180,E1 -3806.001,E2 -3806.001} C_VEL
LIN {X 0,Y 545.086,Z 426.212,A -85,B 0,C 180,E1 -3808.749,E2 -3808.749} C_VEL
LIN {X 0,Y 545.074,Z 426.214,A -85,B 0,C 180,E1 -3811.683,E2 -3811.683} C_VEL
LIN {X 0,Y 545.074,Z 426.216,A -85,B 0,C 180,E1 -3814.564,E2 -3814.564} C_VEL
LIN {X 0,Y 545.061,Z 426.215,A -85,B 0,C 180,E1 -3817.019,E2 -3817.019} C_VEL
LIN {X 0,Y 544.353,Z 426.306,A -85,B 0,C 180,E1 -3817.635,E2 -3817.635} C_VEL
LIN {X 0,Y 541.486,Z 426.663,A -85,B 0,C 180,E1 -3818.636,E2 -3818.636} C_VEL
LIN {X 0,Y 539.098,Z 426.958,A -85,B 0,C 180,E1 -3819.442,E2 -3819.442} C_VEL
LIN {X 0,Y 538.089,Z 427.086,A -85,B 0,C 180,E1 -3820.064,E2 -3820.064} C_VEL
LIN {X 0,Y 538.015,Z 427.09,A -85,B 0,C 180,E1 -3820.274,E2 -3820.274} C_VEL
LIN {X 0,Y 538.032,Z 427.093,A -85,B 0,C 180,E1 -3822.989,E2 -3822.989} C_VEL
LIN {X 0,Y 538.029,Z 427.093,A -85,B 0,C 180,E1 -3825.926,E2 -3825.926} C_VEL
LIN {X 0,Y 538.051,Z 427.088,A -85,B 0,C 180,E1 -3829.253,E2 -3829.253} C_VEL
LIN {X 0,Y 537.994,Z 427.096,A -85,B 0,C 180,E1 -3832.123,E2 -3832.123} C_VEL
LIN {X 0,Y 538.021,Z 427.092,A -85,B 0,C 180,E1 -3834.918,E2 -3834.918} C_VEL
LIN {X 0,Y 538.027,Z 427.092,A -85,B 0,C 180,E1 -3837.619,E2 -3837.619} C_VEL
LIN {X 0,Y 538.045,Z 427.089,A -85,B 0,C 180,E1 -3840.241,E2 -3840.241} C_VEL
LIN {X 0,Y 538.065,Z 427.085,A -85,B 0,C 180,E1 -3842.797,E2 -3842.797} C_VEL
LIN {X 0,Y 538.051,Z 427.09,A -85,B 0,C 180,E1 -3845.293,E2 -3845.293} C_VEL
LIN {X 0,Y 538.026,Z 427.091,A -85,B 0,C 180,E1 -3848.547,E2 -3848.547} C_VEL
LIN {X 0,Y 538.037,Z 427.09,A -85,B 0,C 180,E1 -3850.94,E2 -3850.94} C_VEL
LIN {X 0,Y 538.028,Z 427.094,A -85,B 0,C 180,E1 -3853.299,E2 -3853.299} C_VEL
LIN {X 0,Y 538.068,Z 427.088,A -85,B 0,C 180,E1 -3855.631,E2 -3855.631} C_VEL
LIN {X 0,Y 538.082,Z 427.087,A -85,B 0,C 180,E1 -3858.702,E2 -3858.702} C_VEL
LIN {X 0,Y 538.089,Z 427.085,A -85,B 0,C 180,E1 -3861.74,E2 -3861.74} C_VEL
LIN {X 0,Y 538.162,Z 427.074,A -85,B 0,C 180,E1 -3864.755,E2 -3864.755} C_VEL
LIN {X 0,Y 538.172,Z 427.073,A -85,B 0,C 180,E1 -3867.755,E2 -3867.755} C_VEL
LIN {X 0,Y 538.185,Z 427.072,A -85,B 0,C 180,E1 -3870.748,E2 -3870.748} C_VEL
LIN {X 0,Y 538.141,Z 427.077,A -85,B 0,C 180,E1 -3872.994,E2 -3872.994} C_VEL
LIN {X 0,Y 538.131,Z 427.078,A -85,B 0,C 180,E1 -3875.997,E2 -3875.997} C_VEL
LIN {X 0,Y 538.066,Z 427.087,A -85,B 0,C 180,E1 -3879.017,E2 -3879.017} C_VEL
LIN {X 0,Y 538.087,Z 427.086,A -85,B 0,C 180,E1 -3882.062,E2 -3882.062} C_VEL
LIN {X 0,Y 538.049,Z 427.09,A -85,B 0,C 180,E1 -3885.143,E2 -3885.143} C_VEL
LIN {X 0,Y 538.032,Z 427.089,A -85,B 0,C 180,E1 -3888.27,E2 -3888.27} C_VEL
LIN {X 0,Y 538.04,Z 427.091,A -85,B 0,C 180,E1 -3890.651,E2 -3890.651} C_VEL
LIN {X 0,Y 538.027,Z 427.091,A -85,B 0,C 180,E1 -3893.887,E2 -3893.887} C_VEL
LIN {X 0,Y 538.045,Z 427.089,A -85,B 0,C 180,E1 -3896.366,E2 -3896.366} C_VEL
LIN {X 0,Y 538.034,Z 427.091,A -85,B 0,C 180,E1 -3898.933,E2 -3898.933} C_VEL
LIN {X 0,Y 538.023,Z 427.09,A -85,B 0,C 180,E1 -3901.889,E2 -3901.889} C_VEL
LIN {X 0,Y 537.953,Z 427.103,A -85,B 0,C 180,E1 -3904.177,E2 -3904.177} C_VEL
LIN {X 0,Y 537.8,Z 427.124,A -85,B 0,C 180,E1 -3906.019,E2 -3906.019} C_VEL
LIN {X 0,Y 537.702,Z 427.56,A -85,B 0,C 180,E1 -3907.127,E2 -3907.127} C_VEL
LIN {X 0,Y 537.652,Z 430.23,A -85,B 0,C 180,E1 -3909.829,E2 -3909.829} C_VEL
LIN {X 0,Y 537.661,Z 433.273,A -85,B 0,C 180,E1 -3912.945,E2 -3912.945} C_VEL
LIN {X 0,Y 537.611,Z 436.468,A -85,B 0,C 180,E1 -3916.143,E2 -3916.143} C_VEL
LIN {X 0,Y 537.574,Z 439.488,A -85,B 0,C 180,E1 -3919.18,E2 -3919.18} C_VEL
LIN {X 0,Y 537.499,Z 442.329,A -85,B 0,C 180,E1 -3922.081,E2 -3922.081} C_VEL
LIN {X 0,Y 537.463,Z 445.187,A -85,B 0,C 180,E1 -3924.875,E2 -3924.875} C_VEL
LIN {X 0,Y 537.501,Z 446.398,A -85,B 0,C 180,E1 -3925.973,E2 -3925.973} C_VEL
LIN {X 0,Y 539.968,Z 458.454,A -85,B 0,C 180,E1 -3926.306,E2 -3926.306} C_VEL
LIN {X 0,Y 539.76,Z 471.744,A -85,B 0,C 180,E1 -3926.716,E2 -3926.716} C_VEL
LIN {X 0,Y 539.458,Z 484.964,A -85,B 0,C 180,E1 -3927.271,E2 -3927.271} C_VEL
LIN {X 0,Y 539.158,Z 498.202,A -85,B 0,C 180,E1 -3927.993,E2 -3927.993} C_VEL
LIN {X 0,Y 538.861,Z 509.658,A -85,B 0,C 180,E1 -3928.773,E2 -3928.773} C_VEL
LIN {X 0,Y 538.535,Z 521.294,A -85,B 0,C 180,E1 -3929.736,E2 -3929.736} C_VEL
LIN {X 0,Y 538.292,Z 531.781,A -85,B 0,C 180,E1 -3930.793,E2 -3930.793} C_VEL
LIN {X 0,Y 537.997,Z 541.271,A -85,B 0,C 180,E1 -3931.947,E2 -3931.947} C_VEL
LIN {X 0,Y 537.848,Z 549.75,A -85,B 0,C 180,E1 -3933.204,E2 -3933.204} C_VEL
LIN {X 0,Y 537.715,Z 556.641,A -85,B 0,C 180,E1 -3934.449,E2 -3934.449} C_VEL
LIN {X 0,Y 537.635,Z 562.207,A -85,B 0,C 180,E1 -3935.684,E2 -3935.684} C_VEL
LIN {X 0,Y 537.586,Z 566.578,A -85,B 0,C 180,E1 -3936.908,E2 -3936.908} C_VEL
LIN {X 0,Y 537.545,Z 570.006,A -85,B 0,C 180,E1 -3938.164,E2 -3938.164} C_VEL
LIN {X 0,Y 537.458,Z 572.301,A -85,B 0,C 180,E1 -3939.325,E2 -3939.325} C_VEL
LIN {X 0,Y 537.472,Z 574.097,A -85,B 0,C 180,E1 -3940.919,E2 -3940.919} C_VEL
LIN {X 0,Y 537.476,Z 574.411,A -85,B 0,C 180,E1 -3942.497,E2 -3942.497} C_VEL
LIN {X 0,Y 537.437,Z 573.286,A -85,B 0,C 180,E1 -3944.061,E2 -3944.061} C_VEL
LIN {X 0,Y 537.506,Z 570.725,A -85,B 0,C 180,E1 -3945.615,E2 -3945.615} C_VEL
LIN {X 0,Y 537.573,Z 566.652,A -85,B 0,C 180,E1 -3947.159,E2 -3947.159} C_VEL
LIN {X 0,Y 537.656,Z 560.993,A -85,B 0,C 180,E1 -3948.692,E2 -3948.692} C_VEL
LIN {X 0,Y 537.766,Z 554.623,A -85,B 0,C 180,E1 -3950.028,E2 -3950.028} C_VEL
LIN {X 0,Y 537.925,Z 546.731,A -85,B 0,C 180,E1 -3951.359,E2 -3951.359} C_VEL
LIN {X 0,Y 538.115,Z 538.518,A -85,B 0,C 180,E1 -3952.495,E2 -3952.495} C_VEL
LIN {X 0,Y 538.33,Z 528.681,A -85,B 0,C 180,E1 -3953.629,E2 -3953.629} C_VEL
LIN {X 0,Y 538.626,Z 517.787,A -85,B 0,C 180,E1 -3954.666,E2 -3954.666} C_VEL
LIN {X 0,Y 538.946,Z 505.727,A -85,B 0,C 180,E1 -3955.606,E2 -3955.606} C_VEL
LIN {X 0,Y 539.24,Z 493.858,A -85,B 0,C 180,E1 -3956.357,E2 -3956.357} C_VEL
LIN {X 0,Y 539.552,Z 480.796,A -85,B 0,C 180,E1 -3957.013,E2 -3957.013} C_VEL
LIN {X 0,Y 539.815,Z 467.317,A -85,B 0,C 180,E1 -3957.528,E2 -3957.528} C_VEL
LIN {X 0,Y 539.832,Z 457.696,A -85,B 0,C 180,E1 -3957.808,E2 -3957.808} C_VEL
LIN {X 0,Y 537.481,Z 446.388,A -85,B 0,C 180,E1 -3958.127,E2 -3958.127} C_VEL
LIN {X 0,Y 537.522,Z 443.738,A -85,B 0,C 180,E1 -3960.749,E2 -3960.749} C_VEL
LIN {X 0,Y 537.666,Z 440.939,A -85,B 0,C 180,E1 -3963.747,E2 -3963.747} C_VEL
LIN {X 0,Y 537.725,Z 438.28,A -85,B 0,C 180,E1 -3966.755,E2 -3966.755} C_VEL
LIN {X 0,Y 537.72,Z 436.292,A -85,B 0,C 180,E1 -3969.023,E2 -3969.023} C_VEL
LIN {X 0,Y 537.833,Z 434.1,A -85,B 0,C 180,E1 -3971.471,E2 -3971.471} C_VEL
LIN {X 0,Y 537.854,Z 431.191,A -85,B 0,C 180,E1 -3974.778,E2 -3974.778} C_VEL
LIN {X 0,Y 537.897,Z 428.719,A -85,B 0,C 180,E1 -3977.488,E2 -3977.488} C_VEL
LIN {X 0,Y 537.897,Z 427.309,A -85,B 0,C 180,E1 -3979.065,E2 -3979.065} C_VEL
LIN {X 0,Y 538.004,Z 427.093,A -85,B 0,C 180,E1 -3981.455,E2 -3981.455} C_VEL
LIN {X 0,Y 538.018,Z 427.095,A -85,B 0,C 180,E1 -3983.888,E2 -3983.888} C_VEL
LIN {X 0,Y 538.044,Z 427.092,A -85,B 0,C 180,E1 -3986.366,E2 -3986.366} C_VEL
LIN {X 0,Y 538.051,Z 427.086,A -85,B 0,C 180,E1 -3988.939,E2 -3988.939} C_VEL
LIN {X 0,Y 538.023,Z 427.094,A -85,B 0,C 180,E1 -3991.891,E2 -3991.891} C_VEL
LIN {X 0,Y 538.029,Z 427.089,A -85,B 0,C 180,E1 -3994.622,E2 -3994.622} C_VEL
LIN {X 0,Y 538.003,Z 427.092,A -85,B 0,C 180,E1 -3997.171,E2 -3997.171} C_VEL
LIN {X 0,Y 538.05,Z 427.091,A -85,B 0,C 180,E1 -3999.795,E2 -3999.795} C_VEL
LIN {X 0,Y 538.02,Z 427.091,A -85,B 0,C 180,E1 -4002.786,E2 -4002.786} C_VEL
LIN {X 0,Y 538.026,Z 427.097,A -85,B 0,C 180,E1 -4005.926,E2 -4005.926} C_VEL
LIN {X 0,Y 538.053,Z 427.203,A -85,B 0,C 180,E1 -4008.23,E2 -4008.23} C_VEL
LIN {X 0,Y 538.788,Z 431.35,A -85,B 0,C 180,E1 -4010.318,E2 -4010.318} C_VEL
LIN {X 0,Y 539.037,Z 435.598,A -85,B 0,C 180,E1 -4012.209,E2 -4012.209} C_VEL
LIN {X 0,Y 538.735,Z 443.413,A -85,B 0,C 180,E1 -4015.271,E2 -4015.271} C_VEL
LIN {X 0,Y 538.516,Z 451.138,A -85,B 0,C 180,E1 -4018.027,E2 -4018.027} C_VEL
LIN {X 0,Y 538.331,Z 460.372,A -85,B 0,C 180,E1 -4021.116,E2 -4021.116} C_VEL
LIN {X 0,Y 538.234,Z 468.343,A -85,B 0,C 180,E1 -4023.644,E2 -4023.644} C_VEL
LIN {X 0,Y 538.092,Z 477.696,A -85,B 0,C 180,E1 -4026.525,E2 -4026.525} C_VEL
LIN {X 0,Y 538.002,Z 485.875,A -85,B 0,C 180,E1 -4028.947,E2 -4028.947} C_VEL
LIN {X 0,Y 537.97,Z 493.946,A -85,B 0,C 180,E1 -4031.333,E2 -4031.333} C_VEL
LIN {X 0,Y 537.855,Z 502.186,A -85,B 0,C 180,E1 -4033.855,E2 -4033.855} C_VEL
LIN {X 0,Y 540.039,Z 514.139,A -85,B 0,C 180,E1 -4034.157,E2 -4034.157} C_VEL
LIN {X 0,Y 539.802,Z 528.623,A -85,B 0,C 180,E1 -4034.558,E2 -4034.558} C_VEL
LIN {X 0,Y 539.545,Z 542.17,A -85,B 0,C 180,E1 -4035.093,E2 -4035.093} C_VEL
LIN {X 0,Y 539.26,Z 555.06,A -85,B 0,C 180,E1 -4035.76,E2 -4035.76} C_VEL
LIN {X 0,Y 538.902,Z 568.141,A -85,B 0,C 180,E1 -4036.616,E2 -4036.616} C_VEL
LIN {X 0,Y 538.591,Z 579.888,A -85,B 0,C 180,E1 -4037.567,E2 -4037.567} C_VEL
LIN {X 0,Y 538.353,Z 589.949,A -85,B 0,C 180,E1 -4038.553,E2 -4038.553} C_VEL
LIN {X 0,Y 538.095,Z 599.339,A -85,B 0,C 180,E1 -4039.654,E2 -4039.654} C_VEL
LIN {X 0,Y 537.91,Z 607.407,A -85,B 0,C 180,E1 -4040.79,E2 -4040.79} C_VEL
LIN {X 0,Y 537.763,Z 615.135,A -85,B 0,C 180,E1 -4042.113,E2 -4042.113} C_VEL
LIN {X 0,Y 537.685,Z 621.219,A -85,B 0,C 180,E1 -4043.406,E2 -4043.406} C_VEL
LIN {X 0,Y 537.578,Z 626.201,A -85,B 0,C 180,E1 -4044.749,E2 -4044.749} C_VEL
LIN {X 0,Y 537.576,Z 630.316,A -85,B 0,C 180,E1 -4046.252,E2 -4046.252} C_VEL
LIN {X 0,Y 537.488,Z 633.002,A -85,B 0,C 180,E1 -4047.752,E2 -4047.752} C_VEL
LIN {X 0,Y 537.439,Z 634.333,A -85,B 0,C 180,E1 -4049.251,E2 -4049.251} C_VEL
LIN {X 0,Y 537.439,Z 634.334,A -85,B 0,C 180,E1 -4050.749,E2 -4050.749} C_VEL
LIN {X 0,Y 537.488,Z 633.004,A -85,B 0,C 180,E1 -4052.248,E2 -4052.248} C_VEL
LIN {X 0,Y 537.576,Z 630.32,A -85,B 0,C 180,E1 -4053.748,E2 -4053.748} C_VEL
LIN {X 0,Y 537.579,Z 626.202,A -85,B 0,C 180,E1 -4055.251,E2 -4055.251} C_VEL
LIN {X 0,Y 537.666,Z 620.527,A -85,B 0,C 180,E1 -4056.756,E2 -4056.756} C_VEL
LIN {X 0,Y 537.756,Z 614.128,A -85,B 0,C 180,E1 -4058.076,E2 -4058.076} C_VEL
LIN {X 0,Y 537.97,Z 606.176,A -85,B 0,C 180,E1 -4059.398,E2 -4059.398} C_VEL
LIN {X 0,Y 538.154,Z 597.854,A -85,B 0,C 180,E1 -4060.535,E2 -4060.535} C_VEL
LIN {X 0,Y 538.35,Z 588.677,A -85,B 0,C 180,E1 -4061.584,E2 -4061.584} C_VEL
LIN {X 0,Y 538.669,Z 577.749,A -85,B 0,C 180,E1 -4062.623,E2 -4062.623} C_VEL
LIN {X 0,Y 538.96,Z 565.523,A -85,B 0,C 180,E1 -4063.575,E2 -4063.575} C_VEL
LIN {X 0,Y 539.336,Z 553.406,A -85,B 0,C 180,E1 -4064.334,E2 -4064.334} C_VEL
LIN {X 0,Y 539.571,Z 539.962,A -85,B 0,C 180,E1 -4065.003,E2 -4065.003} C_VEL
LIN {X 0,Y 539.849,Z 525.577,A -85,B 0,C 180,E1 -4065.537,E2 -4065.537} C_VEL
LIN {X 0,Y 539.896,Z 512.432,A -85,B 0,C 180,E1 -4065.883,E2 -4065.883} C_VEL
LIN {X 0,Y 537.855,Z 502.186,A -85,B 0,C 180,E1 -4066.145,E2 -4066.145} C_VEL
LIN {X 0,Y 537.973,Z 492.645,A -85,B 0,C 180,E1 -4069.062,E2 -4069.062} C_VEL
LIN {X 0,Y 538.089,Z 482.027,A -85,B 0,C 180,E1 -4072.257,E2 -4072.257} C_VEL
LIN {X 0,Y 538.23,Z 472.866,A -85,B 0,C 180,E1 -4075.11,E2 -4075.11} C_VEL
LIN {X 0,Y 538.399,Z 463.799,A -85,B 0,C 180,E1 -4078.029,E2 -4078.029} C_VEL
LIN {X 0,Y 538.585,Z 454.781,A -85,B 0,C 180,E1 -4081.026,E2 -4081.026} C_VEL
LIN {X 0,Y 538.772,Z 447.028,A -85,B 0,C 180,E1 -4083.715,E2 -4083.715} C_VEL
LIN {X 0,Y 539.007,Z 439.539,A -85,B 0,C 180,E1 -4086.412,E2 -4086.412} C_VEL
LIN {X 0,Y 539.085,Z 433.377,A -85,B 0,C 180,E1 -4088.738,E2 -4088.738} C_VEL
LIN {X 0,Y 538.052,Z 427.091,A -85,B 0,C 180,E1 -4091.332,E2 -4091.332} C_VEL
LIN {X 0,Y 538.021,Z 427.094,A -85,B 0,C 180,E1 -4094.074,E2 -4094.074} C_VEL
LIN {X 0,Y 538.029,Z 427.09,A -85,B 0,C 180,E1 -4097.011,E2 -4097.011} C_VEL
LIN {X 0,Y 538.047,Z 427.092,A -85,B 0,C 180,E1 -4099.252,E2 -4099.252} C_VEL
LIN {X 0,Y 537.99,Z 427.098,A -85,B 0,C 180,E1 -4102.122,E2 -4102.122} C_VEL
LIN {X 0,Y 538.008,Z 427.095,A -85,B 0,C 180,E1 -4104.916,E2 -4104.916} C_VEL
LIN {X 0,Y 538.027,Z 427.092,A -85,B 0,C 180,E1 -4107.618,E2 -4107.618} C_VEL
LIN {X 0,Y 538.038,Z 427.093,A -85,B 0,C 180,E1 -4110.24,E2 -4110.24} C_VEL
LIN {X 0,Y 538.067,Z 427.089,A -85,B 0,C 180,E1 -4112.796,E2 -4112.796} C_VEL
LIN {X 0,Y 538.044,Z 427.091,A -85,B 0,C 180,E1 -4115.292,E2 -4115.292} C_VEL
LIN {X 0,Y 538.009,Z 427.094,A -85,B 0,C 180,E1 -4118.042,E2 -4118.042} C_VEL
LIN {X 0,Y 538.035,Z 427.093,A -85,B 0,C 180,E1 -4120.94,E2 -4120.94} C_VEL
LIN {X 0,Y 538.022,Z 427.092,A -85,B 0,C 180,E1 -4123.299,E2 -4123.299} C_VEL
LIN {X 0,Y 538.057,Z 427.087,A -85,B 0,C 180,E1 -4125.631,E2 -4125.631} C_VEL
LIN {X 0,Y 538.083,Z 427.084,A -85,B 0,C 180,E1 -4128.702,E2 -4128.702} C_VEL
LIN {X 0,Y 538.085,Z 427.084,A -85,B 0,C 180,E1 -4131.74,E2 -4131.74} C_VEL
LIN {X 0,Y 538.16,Z 427.078,A -85,B 0,C 180,E1 -4134.755,E2 -4134.755} C_VEL
LIN {X 0,Y 538.161,Z 427.077,A -85,B 0,C 180,E1 -4137.755,E2 -4137.755} C_VEL
LIN {X 0,Y 538.179,Z 427.073,A -85,B 0,C 180,E1 -4140.748,E2 -4140.748} C_VEL
LIN {X 0,Y 538.138,Z 427.081,A -85,B 0,C 180,E1 -4142.995,E2 -4142.995} C_VEL
LIN {X 0,Y 538.128,Z 427.082,A -85,B 0,C 180,E1 -4145.997,E2 -4145.997} C_VEL
LIN {X 0,Y 538.071,Z 427.086,A -85,B 0,C 180,E1 -4149.018,E2 -4149.018} C_VEL
LIN {X 0,Y 538.077,Z 427.085,A -85,B 0,C 180,E1 -4152.063,E2 -4152.063} C_VEL
LIN {X 0,Y 538.04,Z 427.091,A -85,B 0,C 180,E1 -4155.144,E2 -4155.144} C_VEL
LIN {X 0,Y 538.029,Z 427.095,A -85,B 0,C 180,E1 -4158.27,E2 -4158.27} C_VEL
LIN {X 0,Y 538.038,Z 427.091,A -85,B 0,C 180,E1 -4160.652,E2 -4160.652} C_VEL
LIN {X 0,Y 538.019,Z 427.095,A -85,B 0,C 180,E1 -4163.888,E2 -4163.888} C_VEL
LIN {X 0,Y 538.038,Z 427.093,A -85,B 0,C 180,E1 -4166.367,E2 -4166.367} C_VEL
LIN {X 0,Y 538.027,Z 427.093,A -85,B 0,C 180,E1 -4168.934,E2 -4168.934} C_VEL
LIN {X 0,Y 538.024,Z 427.094,A -85,B 0,C 180,E1 -4171.891,E2 -4171.891} C_VEL
LIN {X 0,Y 538.024,Z 427.095,A -85,B 0,C 180,E1 -4174.621,E2 -4174.621} C_VEL
LIN {X 0,Y 538.004,Z 427.095,A -85,B 0,C 180,E1 -4177.171,E2 -4177.171} C_VEL
LIN {X 0,Y 538.015,Z 427.09,A -85,B 0,C 180,E1 -4180.274,E2 -4180.274} C_VEL
LIN {X 0,Y 537.367,Z 427.173,A -85,B 0,C 180,E1 -4180.9,E2 -4180.9} C_VEL
LIN {X 0,Y 534.521,Z 427.529,A -85,B 0,C 180,E1 -4181.915,E2 -4181.915} C_VEL
LIN {X 0,Y 532.098,Z 427.832,A -85,B 0,C 180,E1 -4182.732,E2 -4182.732} C_VEL
LIN {X 0,Y 531.051,Z 427.961,A -85,B 0,C 180,E1 -4183.363,E2 -4183.363} C_VEL
LIN {X 0,Y 530.962,Z 427.971,A -85,B 0,C 180,E1 -4183.577,E2 -4183.577} C_VEL
LIN {X 0,Y 530.963,Z 427.971,A -85,B 0,C 180,E1 -4186.506,E2 -4186.506} C_VEL
LIN {X 0,Y 530.991,Z 427.969,A -85,B 0,C 180,E1 -4189.569,E2 -4189.569} C_VEL
LIN {X 0,Y 530.969,Z 427.973,A -85,B 0,C 180,E1 -4192.577,E2 -4192.577} C_VEL
LIN {X 0,Y 531.003,Z 427.969,A -85,B 0,C 180,E1 -4195.312,E2 -4195.312} C_VEL
LIN {X 0,Y 530.972,Z 427.974,A -85,B 0,C 180,E1 -4198.033,E2 -4198.033} C_VEL
LIN {X 0,Y 530.998,Z 427.969,A -85,B 0,C 180,E1 -4200.873,E2 -4200.873} C_VEL
LIN {X 0,Y 531.007,Z 427.966,A -85,B 0,C 180,E1 -4203.257,E2 -4203.257} C_VEL
LIN {X 0,Y 530.988,Z 427.969,A -85,B 0,C 180,E1 -4205.961,E2 -4205.961} C_VEL
LIN {X 0,Y 531.003,Z 427.969,A -85,B 0,C 180,E1 -4209.063,E2 -4209.063} C_VEL
LIN {X 0,Y 531.02,Z 427.963,A -85,B 0,C 180,E1 -4212.278,E2 -4212.278} C_VEL
LIN {X 0,Y 531.023,Z 427.964,A -85,B 0,C 180,E1 -4215.436,E2 -4215.436} C_VEL
LIN {X 0,Y 531.041,Z 427.964,A -85,B 0,C 180,E1 -4218.55,E2 -4218.55} C_VEL
LIN {X 0,Y 531.058,Z 427.961,A -85,B 0,C 180,E1 -4221.63,E2 -4221.63} C_VEL
LIN {X 0,Y 531.121,Z 427.951,A -85,B 0,C 180,E1 -4224.685,E2 -4224.685} C_VEL
LIN {X 0,Y 531.144,Z 427.949,A -85,B 0,C 180,E1 -4227.725,E2 -4227.725} C_VEL
LIN {X 0,Y 531.155,Z 427.947,A -85,B 0,C 180,E1 -4230.758,E2 -4230.758} C_VEL
LIN {X 0,Y 531.108,Z 427.953,A -85,B 0,C 180,E1 -4233.034,E2 -4233.034} C_VEL
LIN {X 0,Y 531.09,Z 427.955,A -85,B 0,C 180,E1 -4236.077,E2 -4236.077} C_VEL
LIN {X 0,Y 531.029,Z 427.965,A -85,B 0,C 180,E1 -4239.138,E2 -4239.138} C_VEL
LIN {X 0,Y 531.044,Z 427.963,A -85,B 0,C 180,E1 -4242.225,E2 -4242.225} C_VEL
LIN {X 0,Y 530.998,Z 427.967,A -85,B 0,C 180,E1 -4245.349,E2 -4245.349} C_VEL
LIN {X 0,Y 530.991,Z 427.967,A -85,B 0,C 180,E1 -4248.521,E2 -4248.521} C_VEL
LIN {X 0,Y 531.002,Z 427.967,A -85,B 0,C 180,E1 -4250.937,E2 -4250.937} C_VEL
LIN {X 0,Y 530.983,Z 427.97,A -85,B 0,C 180,E1 -4254.224,E2 -4254.224} C_VEL
LIN {X 0,Y 531.008,Z 427.966,A -85,B 0,C 180,E1 -4256.743,E2 -4256.743} C_VEL
LIN {X 0,Y 530.985,Z 427.969,A -85,B 0,C 180,E1 -4259.322,E2 -4259.322} C_VEL
LIN {X 0,Y 530.975,Z 427.968,A -85,B 0,C 180,E1 -4262.101,E2 -4262.101} C_VEL
LIN {X 0,Y 530.881,Z 427.986,A -85,B 0,C 180,E1 -4264.837,E2 -4264.837} C_VEL
LIN {X 0,Y 530.692,Z 428.01,A -85,B 0,C 180,E1 -4266.579,E2 -4266.579} C_VEL
LIN {X 0,Y 530.622,Z 428.596,A -85,B 0,C 180,E1 -4267.535,E2 -4267.535} C_VEL
LIN {X 0,Y 530.586,Z 431.466,A -85,B 0,C 180,E1 -4270.468,E2 -4270.468} C_VEL
LIN {X 0,Y 530.571,Z 434.472,A -85,B 0,C 180,E1 -4273.534,E2 -4273.534} C_VEL
LIN {X 0,Y 530.539,Z 437.665,A -85,B 0,C 180,E1 -4276.766,E2 -4276.766} C_VEL
LIN {X 0,Y 530.501,Z 440.405,A -85,B 0,C 180,E1 -4279.522,E2 -4279.522} C_VEL
LIN {X 0,Y 530.412,Z 443.525,A -85,B 0,C 180,E1 -4282.654,E2 -4282.654} C_VEL
LIN {X 0,Y 530.427,Z 446.589,A -85,B 0,C 180,E1 -4285.744,E2 -4285.744} C_VEL
LIN {X 0,Y 533.105,Z 459.825,A -85,B 0,C 180,E1 -4286.134,E2 -4286.134} C_VEL
LIN {X 0,Y 532.9,Z 473.788,A -85,B 0,C 180,E1 -4286.591,E2 -4286.591} C_VEL
LIN {X 0,Y 532.559,Z 487.238,A -85,B 0,C 180,E1 -4287.187,E2 -4287.187} C_VEL
LIN {X 0,Y 532.168,Z 500.72,A -85,B 0,C 180,E1 -4287.965,E2 -4287.965} C_VEL
LIN {X 0,Y 531.827,Z 513.111,A -85,B 0,C 180,E1 -4288.866,E2 -4288.866} C_VEL
LIN {X 0,Y 531.492,Z 524.034,A -85,B 0,C 180,E1 -4289.836,E2 -4289.836} C_VEL
LIN {X 0,Y 531.251,Z 533.957,A -85,B 0,C 180,E1 -4290.897,E2 -4290.897} C_VEL
LIN {X 0,Y 530.912,Z 543.897,A -85,B 0,C 180,E1 -4292.184,E2 -4292.184} C_VEL
LIN {X 0,Y 530.748,Z 551.898,A -85,B 0,C 180,E1 -4293.454,E2 -4293.454} C_VEL
LIN {X 0,Y 530.632,Z 557.73,A -85,B 0,C 180,E1 -4294.577,E2 -4294.577} C_VEL
LIN {X 0,Y 530.524,Z 563.975,A -85,B 0,C 180,E1 -4296.071,E2 -4296.071} C_VEL
LIN {X 0,Y 530.46,Z 568.22,A -85,B 0,C 180,E1 -4297.405,E2 -4297.405} C_VEL
LIN {X 0,Y 530.465,Z 570.268,A -85,B 0,C 180,E1 -4298.225,E2 -4298.225} C_VEL
LIN {X 0,Y 530.349,Z 573.115,A -85,B 0,C 180,E1 -4299.846,E2 -4299.846} C_VEL
LIN {X 0,Y 530.358,Z 574.383,A -85,B 0,C 180,E1 -4301.456,E2 -4301.456} C_VEL
LIN {X 0,Y 530.353,Z 574.182,A -85,B 0,C 180,E1 -4303.05,E2 -4303.05} C_VEL
LIN {X 0,Y 530.337,Z 572.55,A -85,B 0,C 180,E1 -4304.631,E2 -4304.631} C_VEL
LIN {X 0,Y 530.447,Z 569.474,A -85,B 0,C 180,E1 -4306.203,E2 -4306.203} C_VEL
LIN {X 0,Y 530.516,Z 564.91,A -85,B 0,C 180,E1 -4307.763,E2 -4307.763} C_VEL
LIN {X 0,Y 530.608,Z 560.277,A -85,B 0,C 180,E1 -4308.951,E2 -4308.951} C_VEL
LIN {X 0,Y 530.713,Z 553.864,A -85,B 0,C 180,E1 -4310.279,E2 -4310.279} C_VEL
LIN {X 0,Y 530.874,Z 545.814,A -85,B 0,C 180,E1 -4311.626,E2 -4311.626} C_VEL
LIN {X 0,Y 531.175,Z 536.526,A -85,B 0,C 180,E1 -4312.889,E2 -4312.889} C_VEL
LIN {X 0,Y 531.387,Z 527.348,A -85,B 0,C 180,E1 -4313.926,E2 -4313.926} C_VEL
LIN {X 0,Y 531.731,Z 516.125,A -85,B 0,C 180,E1 -4314.976,E2 -4314.976} C_VEL
LIN {X 0,Y 532.041,Z 505.032,A -85,B 0,C 180,E1 -4315.833,E2 -4315.833} C_VEL
LIN {X 0,Y 532.352,Z 493.001,A -85,B 0,C 180,E1 -4316.594,E2 -4316.594} C_VEL
LIN {X 0,Y 532.74,Z 479.651,A -85,B 0,C 180,E1 -4317.259,E2 -4317.259} C_VEL
LIN {X 0,Y 533.037,Z 465.785,A -85,B 0,C 180,E1 -4317.78,E2 -4317.78} C_VEL
LIN {X 0,Y 532.905,Z 458.273,A -85,B 0,C 180,E1 -4318.004,E2 -4318.004} C_VEL
LIN {X 0,Y 530.41,Z 446.686,A -85,B 0,C 180,E1 -4318.339,E2 -4318.339} C_VEL
LIN {X 0,Y 530.451,Z 444.368,A -85,B 0,C 180,E1 -4320.759,E2 -4320.759} C_VEL
LIN {X 0,Y 530.615,Z 441.58,A -85,B 0,C 180,E1 -4323.797,E2 -4323.797} C_VEL
LIN {X 0,Y 530.665,Z 438.972,A -85,B 0,C 180,E1 -4326.845,E2 -4326.845} C_VEL
LIN {X 0,Y 530.663,Z 436.934,A -85,B 0,C 180,E1 -4329.144,E2 -4329.144} C_VEL
LIN {X 0,Y 530.777,Z 434.832,A -85,B 0,C 180,E1 -4331.532,E2 -4331.532} C_VEL
LIN {X 0,Y 530.806,Z 431.881,A -85,B 0,C 180,E1 -4334.868,E2 -4334.868} C_VEL
LIN {X 0,Y 530.833,Z 429.333,A -85,B 0,C 180,E1 -4337.729,E2 -4337.729} C_VEL
LIN {X 0,Y 530.864,Z 427.988,A -85,B 0,C 180,E1 -4339.328,E2 -4339.328} C_VEL
LIN {X 0,Y 530.971,Z 427.974,A -85,B 0,C 180,E1 -4342.103,E2 -4342.103} C_VEL
LIN {X 0,Y 531.002,Z 427.964,A -85,B 0,C 180,E1 -4345.058,E2 -4345.058} C_VEL
LIN {X 0,Y 531.012,Z 427.965,A -85,B 0,C 180,E1 -4347.596,E2 -4347.596} C_VEL
LIN {X 0,Y 530.977,Z 427.969,A -85,B 0,C 180,E1 -4350.647,E2 -4350.647} C_VEL
LIN {X 0,Y 530.988,Z 427.971,A -85,B 0,C 180,E1 -4353.773,E2 -4353.773} C_VEL
LIN {X 0,Y 530.964,Z 427.97,A -85,B 0,C 180,E1 -4356.558,E2 -4356.558} C_VEL
LIN {X 0,Y 531.002,Z 427.97,A -85,B 0,C 180,E1 -4359.858,E2 -4359.858} C_VEL
LIN {X 0,Y 530.979,Z 427.97,A -85,B 0,C 180,E1 -4362.457,E2 -4362.457} C_VEL
LIN {X 0,Y 530.985,Z 427.973,A -85,B 0,C 180,E1 -4365.621,E2 -4365.621} C_VEL
LIN {X 0,Y 531.006,Z 428.049,A -85,B 0,C 180,E1 -4367.832,E2 -4367.832} C_VEL
LIN {X 0,Y 531.775,Z 432.26,A -85,B 0,C 180,E1 -4370.044,E2 -4370.044} C_VEL
LIN {X 0,Y 532.083,Z 435.642,A -85,B 0,C 180,E1 -4371.626,E2 -4371.626} C_VEL
LIN {X 0,Y 531.901,Z 440.668,A -85,B 0,C 180,E1 -4373.706,E2 -4373.706} C_VEL
LIN {X 0,Y 531.605,Z 447.688,A -85,B 0,C 180,E1 -4376.396,E2 -4376.396} C_VEL
LIN {X 0,Y 531.428,Z 454.905,A -85,B 0,C 180,E1 -4378.952,E2 -4378.952} C_VEL
LIN {X 0,Y 531.292,Z 462.665,A -85,B 0,C 180,E1 -4381.562,E2 -4381.562} C_VEL
LIN {X 0,Y 531.141,Z 471.978,A -85,B 0,C 180,E1 -4384.539,E2 -4384.539} C_VEL
LIN {X 0,Y 531.032,Z 481.349,A -85,B 0,C 180,E1 -4387.431,E2 -4387.431} C_VEL
LIN {X 0,Y 530.915,Z 492.211,A -85,B 0,C 180,E1 -4390.675,E2 -4390.675} C_VEL
LIN {X 0,Y 530.813,Z 502.185,A -85,B 0,C 180,E1 -4393.635,E2 -4393.635} C_VEL
LIN {X 0,Y 533.224,Z 514.918,A -85,B 0,C 180,E1 -4393.966,E2 -4393.966} C_VEL
LIN {X 0,Y 532.965,Z 528.623,A -85,B 0,C 180,E1 -4394.355,E2 -4394.355} C_VEL
LIN {X 0,Y 532.675,Z 542.169,A -85,B 0,C 180,E1 -4394.896,E2 -4394.896} C_VEL
LIN {X 0,Y 532.368,Z 555.058,A -85,B 0,C 180,E1 -4395.572,E2 -4395.572} C_VEL
LIN {X 0,Y 531.994,Z 566.848,A -85,B 0,C 180,E1 -4396.341,E2 -4396.341} C_VEL
LIN {X 0,Y 531.676,Z 578.818,A -85,B 0,C 180,E1 -4397.305,E2 -4397.305} C_VEL
LIN {X 0,Y 531.343,Z 590.258,A -85,B 0,C 180,E1 -4398.433,E2 -4398.433} C_VEL
LIN {X 0,Y 531.087,Z 599.339,A -85,B 0,C 180,E1 -4399.516,E2 -4399.516} C_VEL
LIN {X 0,Y 530.886,Z 607.406,A -85,B 0,C 180,E1 -4400.667,E2 -4400.667} C_VEL
LIN {X 0,Y 530.684,Z 615.135,A -85,B 0,C 180,E1 -4402.007,E2 -4402.007} C_VEL
LIN {X 0,Y 530.61,Z 621.593,A -85,B 0,C 180,E1 -4403.406,E2 -4403.406} C_VEL
LIN {X 0,Y 530.514,Z 626.201,A -85,B 0,C 180,E1 -4404.679,E2 -4404.679} C_VEL
LIN {X 0,Y 530.497,Z 630.317,A -85,B 0,C 180,E1 -4406.202,E2 -4406.202} C_VEL
LIN {X 0,Y 530.409,Z 633.002,A -85,B 0,C 180,E1 -4407.722,E2 -4407.722} C_VEL
LIN {X 0,Y 530.341,Z 634.333,A -85,B 0,C 180,E1 -4409.241,E2 -4409.241} C_VEL
LIN {X 0,Y 530.341,Z 634.334,A -85,B 0,C 180,E1 -4410.759,E2 -4410.759} C_VEL
LIN {X 0,Y 530.409,Z 633.005,A -85,B 0,C 180,E1 -4412.278,E2 -4412.278} C_VEL
LIN {X 0,Y 530.497,Z 630.32,A -85,B 0,C 180,E1 -4413.798,E2 -4413.798} C_VEL
LIN {X 0,Y 530.515,Z 626.202,A -85,B 0,C 180,E1 -4415.321,E2 -4415.321} C_VEL
LIN {X 0,Y 530.573,Z 620.527,A -85,B 0,C 180,E1 -4416.847,E2 -4416.847} C_VEL
LIN {X 0,Y 530.709,Z 614.128,A -85,B 0,C 180,E1 -4418.184,E2 -4418.184} C_VEL
LIN {X 0,Y 530.927,Z 606.175,A -85,B 0,C 180,E1 -4419.524,E2 -4419.524} C_VEL
LIN {X 0,Y 531.13,Z 597.854,A -85,B 0,C 180,E1 -4420.676,E2 -4420.676} C_VEL
LIN {X 0,Y 531.454,Z 587.356,A -85,B 0,C 180,E1 -4421.879,E2 -4421.879} C_VEL
LIN {X 0,Y 531.718,Z 576.65,A -85,B 0,C 180,E1 -4422.888,E2 -4422.888} C_VEL
LIN {X 0,Y 532.104,Z 564.104,A -85,B 0,C 180,E1 -4423.851,E2 -4423.851} C_VEL
LIN {X 0,Y 532.491,Z 551.643,A -85,B 0,C 180,E1 -4424.62,E2 -4424.62} C_VEL
LIN {X 0,Y 532.757,Z 538.83,A -85,B 0,C 180,E1 -4425.248,E2 -4425.248} C_VEL
LIN {X 0,Y 533.035,Z 524.416,A -85,B 0,C 180,E1 -4425.778,E2 -4425.778} C_VEL
LIN {X 0,Y 533.114,Z 513.714,A -85,B 0,C 180,E1 -4426.063,E2 -4426.063} C_VEL
LIN {X 0,Y 530.813,Z 502.185,A -85,B 0,C 180,E1 -4426.365,E2 -4426.365} C_VEL
LIN {X 0,Y 530.915,Z 492.375,A -85,B 0,C 180,E1 -4429.325,E2 -4429.325} C_VEL
LIN {X 0,Y 531.044,Z 481.751,A -85,B 0,C 180,E1 -4432.569,E2 -4432.569} C_VEL
LIN {X 0,Y 531.232,Z 472.682,A -85,B 0,C 180,E1 -4435.465,E2 -4435.465} C_VEL
LIN {X 0,Y 531.39,Z 463.622,A -85,B 0,C 180,E1 -4438.432,E2 -4438.432} C_VEL
LIN {X 0,Y 531.588,Z 455.934,A -85,B 0,C 180,E1 -4441.038,E2 -4441.038} C_VEL
LIN {X 0,Y 531.858,Z 447.067,A -85,B 0,C 180,E1 -4444.166,E2 -4444.166} C_VEL
LIN {X 0,Y 532.086,Z 439.525,A -85,B 0,C 180,E1 -4446.939,E2 -4446.939} C_VEL
LIN {X 0,Y 532.131,Z 434.673,A -85,B 0,C 180,E1 -4448.81,E2 -4448.81} C_VEL
LIN {X 0,Y 531.019,Z 427.968,A -85,B 0,C 180,E1 -4451.606,E2 -4451.606} C_VEL
LIN {X 0,Y 530.983,Z 427.97,A -85,B 0,C 180,E1 -4454.546,E2 -4454.546} C_VEL
LIN {X 0,Y 530.985,Z 427.971,A -85,B 0,C 180,E1 -4457.833,E2 -4457.833} C_VEL
LIN {X 0,Y 530.986,Z 427.972,A -85,B 0,C 180,E1 -4460.557,E2 -4460.557} C_VEL
LIN {X 0,Y 530.964,Z 427.97,A -85,B 0,C 180,E1 -4463.843,E2 -4463.843} C_VEL
LIN {X 0,Y 530.994,Z 427.968,A -85,B 0,C 180,E1 -4466.494,E2 -4466.494} C_VEL
LIN {X 0,Y 530.977,Z 427.969,A -85,B 0,C 180,E1 -4469.353,E2 -4469.353} C_VEL
LIN {X 0,Y 531.012,Z 427.965,A -85,B 0,C 180,E1 -4472.404,E2 -4472.404} C_VEL
LIN {X 0,Y 531.002,Z 427.966,A -85,B 0,C 180,E1 -4474.942,E2 -4474.942} C_VEL
LIN {X 0,Y 530.965,Z 427.973,A -85,B 0,C 180,E1 -4478.247,E2 -4478.247} C_VEL
LIN {X 0,Y 530.991,Z 427.968,A -85,B 0,C 180,E1 -4480.677,E2 -4480.677} C_VEL
LIN {X 0,Y 530.987,Z 427.968,A -85,B 0,C 180,E1 -4483.071,E2 -4483.071} C_VEL
LIN {X 0,Y 531.012,Z 427.966,A -85,B 0,C 180,E1 -4485.436,E2 -4485.436} C_VEL
LIN {X 0,Y 531.04,Z 427.962,A -85,B 0,C 180,E1 -4488.55,E2 -4488.55} C_VEL
LIN {X 0,Y 531.054,Z 427.96,A -85,B 0,C 180,E1 -4491.63,E2 -4491.63} C_VEL
LIN {X 0,Y 531.118,Z 427.954,A -85,B 0,C 180,E1 -4494.685,E2 -4494.685} C_VEL
LIN {X 0,Y 531.133,Z 427.952,A -85,B 0,C 180,E1 -4497.725,E2 -4497.725} C_VEL
LIN {X 0,Y 531.148,Z 427.949,A -85,B 0,C 180,E1 -4500.758,E2 -4500.758} C_VEL
LIN {X 0,Y 531.104,Z 427.957,A -85,B 0,C 180,E1 -4503.034,E2 -4503.034} C_VEL
LIN {X 0,Y 531.086,Z 427.958,A -85,B 0,C 180,E1 -4506.077,E2 -4506.077} C_VEL
LIN {X 0,Y 531.03,Z 427.962,A -85,B 0,C 180,E1 -4509.138,E2 -4509.138} C_VEL
LIN {X 0,Y 531.035,Z 427.963,A -85,B 0,C 180,E1 -4512.225,E2 -4512.225} C_VEL
LIN {X 0,Y 530.99,Z 427.97,A -85,B 0,C 180,E1 -4515.35,E2 -4515.35} C_VEL
LIN {X 0,Y 531.011,Z 427.965,A -85,B 0,C 180,E1 -4517.723,E2 -4517.723} C_VEL
LIN {X 0,Y 530.997,Z 427.97,A -85,B 0,C 180,E1 -4520.938,E2 -4520.938} C_VEL
LIN {X 0,Y 530.975,Z 427.97,A -85,B 0,C 180,E1 -4524.225,E2 -4524.225} C_VEL
LIN {X 0,Y 531.001,Z 427.967,A -85,B 0,C 180,E1 -4526.744,E2 -4526.744} C_VEL
LIN {X 0,Y 530.978,Z 427.972,A -85,B 0,C 180,E1 -4529.323,E2 -4529.323} C_VEL
LIN {X 0,Y 530.977,Z 427.972,A -85,B 0,C 180,E1 -4532.104,E2 -4532.104} C_VEL
LIN {X 0,Y 530.981,Z 427.971,A -85,B 0,C 180,E1 -4534.854,E2 -4534.854} C_VEL
LIN {X 0,Y 530.963,Z 427.974,A -85,B 0,C 180,E1 -4537.508,E2 -4537.508} C_VEL
LIN {X 0,Y 530.978,Z 427.97,A -85,B 0,C 180,E1 -4540.434,E2 -4540.434} C_VEL
LIN {X 0,Y 530.966,Z 427.971,A -85,B 0,C 180,E1 -4543.495,E2 -4543.495} C_VEL
LIN {X 0,Y 530.962,Z 427.971,A -85,B 0,C 180,E1 -4543.577,E2 -4543.577} C_VEL
LIN {X 0,Y 530.289,Z 428.058,A -85,B 0,C 180,E1 -4544.21,E2 -4544.21} C_VEL
LIN {X 0,Y 527.44,Z 428.412,A -85,B 0,C 180,E1 -4545.239,E2 -4545.239} C_VEL
LIN {X 0,Y 525.036,Z 428.713,A -85,B 0,C 180,E1 -4546.068,E2 -4546.068} C_VEL
LIN {X 0,Y 524.002,Z 428.841,A -85,B 0,C 180,E1 -4546.707,E2 -4546.707} C_VEL
LIN {X 0,Y 523.917,Z 428.85,A -85,B 0,C 180,E1 -4546.924,E2 -4546.924} C_VEL
LIN {X 0,Y 523.963,Z 428.846,A -85,B 0,C 180,E1 -4549.923,E2 -4549.923} C_VEL
LIN {X 0,Y 523.912,Z 428.851,A -85,B 0,C 180,E1 -4552.869,E2 -4552.869} C_VEL
LIN {X 0,Y 523.945,Z 428.846,A -85,B 0,C 180,E1 -4555.711,E2 -4555.711} C_VEL
LIN {X 0,Y 523.926,Z 428.847,A -85,B 0,C 180,E1 -4558.457,E2 -4558.457} C_VEL
LIN {X 0,Y 523.946,Z 428.847,A -85,B 0,C 180,E1 -4561.126,E2 -4561.126} C_VEL
LIN {X 0,Y 523.987,Z 428.841,A -85,B 0,C 180,E1 -4563.981,E2 -4563.981} C_VEL
LIN {X 0,Y 523.929,Z 428.85,A -85,B 0,C 180,E1 -4566.271,E2 -4566.271} C_VEL
LIN {X 0,Y 523.949,Z 428.846,A -85,B 0,C 180,E1 -4568.767,E2 -4568.767} C_VEL
LIN {X 0,Y 523.953,Z 428.844,A -85,B 0,C 180,E1 -4571.221,E2 -4571.221} C_VEL
LIN {X 0,Y 523.94,Z 428.847,A -85,B 0,C 180,E1 -4573.639,E2 -4573.639} C_VEL
LIN {X 0,Y 523.944,Z 428.847,A -85,B 0,C 180,E1 -4576.028,E2 -4576.028} C_VEL
LIN {X 0,Y 524.017,Z 428.838,A -85,B 0,C 180,E1 -4578.394,E2 -4578.394} C_VEL
LIN {X 0,Y 524.006,Z 428.841,A -85,B 0,C 180,E1 -4581.516,E2 -4581.516} C_VEL
LIN {X 0,Y 524.082,Z 428.829,A -85,B 0,C 180,E1 -4584.614,E2 -4584.614} C_VEL
LIN {X 0,Y 524.116,Z 428.824,A -85,B 0,C 180,E1 -4587.695,E2 -4587.695} C_VEL
LIN {X 0,Y 524.126,Z 428.823,A -85,B 0,C 180,E1 -4590.768,E2 -4590.768} C_VEL
LIN {X 0,Y 524.075,Z 428.829,A -85,B 0,C 180,E1 -4593.075,E2 -4593.075} C_VEL
LIN {X 0,Y 524.053,Z 428.833,A -85,B 0,C 180,E1 -4596.159,E2 -4596.159} C_VEL
LIN {X 0,Y 523.998,Z 428.842,A -85,B 0,C 180,E1 -4599.262,E2 -4599.262} C_VEL
LIN {X 0,Y 524.007,Z 428.839,A -85,B 0,C 180,E1 -4601.739,E2 -4601.739} C_VEL
LIN {X 0,Y 523.997,Z 428.841,A -85,B 0,C 180,E1 -4605.052,E2 -4605.052} C_VEL
LIN {X 0,Y 523.967,Z 428.842,A -85,B 0,C 180,E1 -4607.969,E2 -4607.969} C_VEL
LIN {X 0,Y 523.975,Z 428.844,A -85,B 0,C 180,E1 -4610.41,E2 -4610.41} C_VEL
LIN {X 0,Y 523.92,Z 428.851,A -85,B 0,C 180,E1 -4612.893,E2 -4612.893} C_VEL
LIN {X 0,Y 523.956,Z 428.845,A -85,B 0,C 180,E1 -4615.418,E2 -4615.418} C_VEL
LIN {X 0,Y 523.972,Z 428.841,A -85,B 0,C 180,E1 -4617.998,E2 -4617.998} C_VEL
LIN {X 0,Y 523.948,Z 428.846,A -85,B 0,C 180,E1 -4620.855,E2 -4620.855} C_VEL
LIN {X 0,Y 523.911,Z 428.851,A -85,B 0,C 180,E1 -4623.726,E2 -4623.726} C_VEL
LIN {X 0,Y 523.685,Z 428.882,A -85,B 0,C 180,E1 -4626.368,E2 -4626.368} C_VEL
LIN {X 0,Y 523.56,Z 428.897,A -85,B 0,C 180,E1 -4627.16,E2 -4627.16} C_VEL
LIN {X 0,Y 523.536,Z 431.752,A -85,B 0,C 180,E1 -4630.117,E2 -4630.117} C_VEL
LIN {X 0,Y 523.506,Z 434.773,A -85,B 0,C 180,E1 -4633.209,E2 -4633.209} C_VEL
LIN {X 0,Y 523.487,Z 437.955,A -85,B 0,C 180,E1 -4636.465,E2 -4636.465} C_VEL
LIN {X 0,Y 523.416,Z 441.324,A -85,B 0,C 180,E1 -4639.871,E2 -4639.871} C_VEL
LIN {X 0,Y 523.326,Z 444.254,A -85,B 0,C 180,E1 -4642.819,E2 -4642.819} C_VEL
LIN {X 0,Y 523.341,Z 446.969,A -85,B 0,C 180,E1 -4645.53,E2 -4645.53} C_VEL
LIN {X 0,Y 526.277,Z 460.299,A -85,B 0,C 180,E1 -4645.931,E2 -4645.931} C_VEL
LIN {X 0,Y 526.034,Z 474.571,A -85,B 0,C 180,E1 -4646.407,E2 -4646.407} C_VEL
LIN {X 0,Y 525.649,Z 488.575,A -85,B 0,C 180,E1 -4647.047,E2 -4647.047} C_VEL
LIN {X 0,Y 525.292,Z 500.613,A -85,B 0,C 180,E1 -4647.758,E2 -4647.758} C_VEL
LIN {X 0,Y 524.906,Z 512.938,A -85,B 0,C 180,E1 -4648.664,E2 -4648.664} C_VEL
LIN {X 0,Y 524.5,Z 524.643,A -85,B 0,C 180,E1 -4649.725,E2 -4649.725} C_VEL
LIN {X 0,Y 524.233,Z 534.465,A -85,B 0,C 180,E1 -4650.806,E2 -4650.806} C_VEL
LIN {X 0,Y 523.873,Z 543.514,A -85,B 0,C 180,E1 -4651.995,E2 -4651.995} C_VEL
LIN {X 0,Y 523.709,Z 551.59,A -85,B 0,C 180,E1 -4653.284,E2 -4653.284} C_VEL
LIN {X 0,Y 523.55,Z 558.124,A -85,B 0,C 180,E1 -4654.56,E2 -4654.56} C_VEL
LIN {X 0,Y 523.436,Z 563.729,A -85,B 0,C 180,E1 -4655.923,E2 -4655.923} C_VEL
LIN {X 0,Y 523.363,Z 568.653,A -85,B 0,C 180,E1 -4657.498,E2 -4657.498} C_VEL
LIN {X 0,Y 523.303,Z 571.41,A -85,B 0,C 180,E1 -4658.739,E2 -4658.739} C_VEL
LIN {X 0,Y 523.288,Z 573.708,A -85,B 0,C 180,E1 -4660.381,E2 -4660.381} C_VEL
LIN {X 0,Y 523.253,Z 574.497,A -85,B 0,C 180,E1 -4662.006,E2 -4662.006} C_VEL
LIN {X 0,Y 523.28,Z 574.334,A -85,B 0,C 180,E1 -4662.814,E2 -4662.814} C_VEL
LIN {X 0,Y 523.237,Z 572.913,A -85,B 0,C 180,E1 -4664.417,E2 -4664.417} C_VEL
LIN {X 0,Y 523.328,Z 570.048,A -85,B 0,C 180,E1 -4666.011,E2 -4666.011} C_VEL
LIN {X 0,Y 523.427,Z 565.699,A -85,B 0,C 180,E1 -4667.594,E2 -4667.594} C_VEL
LIN {X 0,Y 523.51,Z 561.063,A -85,B 0,C 180,E1 -4668.856,E2 -4668.856} C_VEL
LIN {X 0,Y 523.645,Z 554.119,A -85,B 0,C 180,E1 -4670.342,E2 -4670.342} C_VEL
LIN {X 0,Y 523.839,Z 546.123,A -85,B 0,C 180,E1 -4671.707,E2 -4671.707} C_VEL
LIN {X 0,Y 524.108,Z 537.77,A -85,B 0,C 180,E1 -4672.876,E2 -4672.876} C_VEL
LIN {X 0,Y 524.407,Z 527.863,A -85,B 0,C 180,E1 -4674.038,E2 -4674.038} C_VEL
LIN {X 0,Y 524.79,Z 516.835,A -85,B 0,C 180,E1 -4675.102,E2 -4675.102} C_VEL
LIN {X 0,Y 525.123,Z 505.914,A -85,B 0,C 180,E1 -4675.971,E2 -4675.971} C_VEL
LIN {X 0,Y 525.474,Z 494.072,A -85,B 0,C 180,E1 -4676.741,E2 -4676.741} C_VEL
LIN {X 0,Y 525.844,Z 481.003,A -85,B 0,C 180,E1 -4677.414,E2 -4677.414} C_VEL
LIN {X 0,Y 526.173,Z 467.469,A -85,B 0,C 180,E1 -4677.943,E2 -4677.943} C_VEL
LIN {X 0,Y 526.13,Z 459.685,A -85,B 0,C 180,E1 -4678.182,E2 -4678.182} C_VEL
LIN {X 0,Y 523.357,Z 447.218,A -85,B 0,C 180,E1 -4678.557,E2 -4678.557} C_VEL
LIN {X 0,Y 523.392,Z 444.421,A -85,B 0,C 180,E1 -4681.539,E2 -4681.539} C_VEL
LIN {X 0,Y 523.551,Z 441.682,A -85,B 0,C 180,E1 -4684.62,E2 -4684.62} C_VEL
LIN {X 0,Y 523.616,Z 439.643,A -85,B 0,C 180,E1 -4686.938,E2 -4686.938} C_VEL
LIN {X 0,Y 523.616,Z 437.602,A -85,B 0,C 180,E1 -4689.269,E2 -4689.269} C_VEL
LIN {X 0,Y 523.713,Z 435.541,A -85,B 0,C 180,E1 -4691.612,E2 -4691.612} C_VEL
LIN {X 0,Y 523.754,Z 432.665,A -85,B 0,C 180,E1 -4694.958,E2 -4694.958} C_VEL
LIN {X 0,Y 523.812,Z 430.021,A -85,B 0,C 180,E1 -4697.974,E2 -4697.974} C_VEL
LIN {X 0,Y 523.858,Z 428.86,A -85,B 0,C 180,E1 -4699.597,E2 -4699.597} C_VEL
LIN {X 0,Y 523.914,Z 428.853,A -85,B 0,C 180,E1 -4702.244,E2 -4702.244} C_VEL
LIN {X 0,Y 523.931,Z 428.849,A -85,B 0,C 180,E1 -4704.572,E2 -4704.572} C_VEL
LIN {X 0,Y 523.952,Z 428.842,A -85,B 0,C 180,E1 -4707.133,E2 -4707.133} C_VEL
LIN {X 0,Y 523.951,Z 428.846,A -85,B 0,C 180,E1 -4709.755,E2 -4709.755} C_VEL
LIN {X 0,Y 523.935,Z 428.847,A -85,B 0,C 180,E1 -4712.449,E2 -4712.449} C_VEL
LIN {X 0,Y 523.931,Z 428.845,A -85,B 0,C 180,E1 -4715.226,E2 -4715.226} C_VEL
LIN {X 0,Y 523.913,Z 428.853,A -85,B 0,C 180,E1 -4718.102,E2 -4718.102} C_VEL
LIN {X 0,Y 523.958,Z 428.842,A -85,B 0,C 180,E1 -4721.091,E2 -4721.091} C_VEL
LIN {X 0,Y 523.938,Z 428.851,A -85,B 0,C 180,E1 -4724.228,E2 -4724.228} C_VEL
LIN {X 0,Y 523.945,Z 428.866,A -85,B 0,C 180,E1 -4727.389,E2 -4727.389} C_VEL
LIN {X 0,Y 524.846,Z 433.649,A -85,B 0,C 180,E1 -4730.004,E2 -4730.004} C_VEL
LIN {X 0,Y 525.123,Z 436.824,A -85,B 0,C 180,E1 -4731.514,E2 -4731.514} C_VEL
LIN {X 0,Y 524.884,Z 442.489,A -85,B 0,C 180,E1 -4733.905,E2 -4733.905} C_VEL
LIN {X 0,Y 524.631,Z 448.302,A -85,B 0,C 180,E1 -4736.156,E2 -4736.156} C_VEL
LIN {X 0,Y 524.504,Z 454.68,A -85,B 0,C 180,E1 -4738.496,E2 -4738.496} C_VEL
LIN {X 0,Y 524.267,Z 463.656,A -85,B 0,C 180,E1 -4741.583,E2 -4741.583} C_VEL
LIN {X 0,Y 524.073,Z 472.898,A -85,B 0,C 180,E1 -4744.588,E2 -4744.588} C_VEL
LIN {X 0,Y 523.953,Z 482.996,A -85,B 0,C 180,E1 -4747.748,E2 -4747.748} C_VEL
LIN {X 0,Y 523.814,Z 493.122,A -85,B 0,C 180,E1 -4750.81,E2 -4750.81} C_VEL
LIN {X 0,Y 523.738,Z 501.868,A -85,B 0,C 180,E1 -4753.432,E2 -4753.432} C_VEL
LIN {X 0,Y 526.375,Z 516.146,A -85,B 0,C 180,E1 -4753.791,E2 -4753.791} C_VEL
LIN {X 0,Y 526.1,Z 529.473,A -85,B 0,C 180,E1 -4754.187,E2 -4754.187} C_VEL
LIN {X 0,Y 525.759,Z 542.992,A -85,B 0,C 180,E1 -4754.742,E2 -4754.742} C_VEL
LIN {X 0,Y 525.418,Z 556.609,A -85,B 0,C 180,E1 -4755.475,E2 -4755.475} C_VEL
LIN {X 0,Y 525.013,Z 569.428,A -85,B 0,C 180,E1 -4756.354,E2 -4756.354} C_VEL
LIN {X 0,Y 524.627,Z 580.954,A -85,B 0,C 180,E1 -4757.329,E2 -4757.329} C_VEL
LIN {X 0,Y 524.311,Z 591.394,A -85,B 0,C 180,E1 -4758.401,E2 -4758.401} C_VEL
LIN {X 0,Y 524.009,Z 600.823,A -85,B 0,C 180,E1 -4759.569,E2 -4759.569} C_VEL
LIN {X 0,Y 523.753,Z 609.803,A -85,B 0,C 180,E1 -4760.929,E2 -4760.929} C_VEL
LIN {X 0,Y 523.569,Z 617.055,A -85,B 0,C 180,E1 -4762.286,E2 -4762.286} C_VEL
LIN {X 0,Y 523.473,Z 623.569,A -85,B 0,C 180,E1 -4763.834,E2 -4763.834} C_VEL
LIN {X 0,Y 523.376,Z 627.38,A -85,B 0,C 180,E1 -4764.993,E2 -4764.993} C_VEL
LIN {X 0,Y 523.419,Z 630.316,A -85,B 0,C 180,E1 -4766.151,E2 -4766.151} C_VEL
LIN {X 0,Y 523.333,Z 633.002,A -85,B 0,C 180,E1 -4767.691,E2 -4767.691} C_VEL
LIN {X 0,Y 523.247,Z 634.334,A -85,B 0,C 180,E1 -4769.23,E2 -4769.23} C_VEL
LIN {X 0,Y 523.247,Z 634.334,A -85,B 0,C 180,E1 -4770.77,E2 -4770.77} C_VEL
LIN {X 0,Y 523.333,Z 633.005,A -85,B 0,C 180,E1 -4772.309,E2 -4772.309} C_VEL
LIN {X 0,Y 523.419,Z 630.32,A -85,B 0,C 180,E1 -4773.849,E2 -4773.849} C_VEL
LIN {X 0,Y 523.452,Z 626.202,A -85,B 0,C 180,E1 -4775.393,E2 -4775.393} C_VEL
LIN {X 0,Y 523.494,Z 620.527,A -85,B 0,C 180,E1 -4776.94,E2 -4776.94} C_VEL
LIN {X 0,Y 523.664,Z 614.128,A -85,B 0,C 180,E1 -4778.295,E2 -4778.295} C_VEL
LIN {X 0,Y 523.862,Z 606.175,A -85,B 0,C 180,E1 -4779.654,E2 -4779.654} C_VEL
LIN {X 0,Y 524.117,Z 597.853,A -85,B 0,C 180,E1 -4780.82,E2 -4780.82} C_VEL
LIN {X 0,Y 524.448,Z 587.091,A -85,B 0,C 180,E1 -4782.068,E2 -4782.068} C_VEL
LIN {X 0,Y 524.774,Z 576.651,A -85,B 0,C 180,E1 -4783.061,E2 -4783.061} C_VEL
LIN {X 0,Y 525.189,Z 564.103,A -85,B 0,C 180,E1 -4784.037,E2 -4784.037} C_VEL
LIN {X 0,Y 525.619,Z 551.575,A -85,B 0,C 180,E1 -4784.816,E2 -4784.816} C_VEL
LIN {X 0,Y 525.91,Z 538.663,A -85,B 0,C 180,E1 -4785.452,E2 -4785.452} C_VEL
LIN {X 0,Y 526.217,Z 524.154,A -85,B 0,C 180,E1 -4785.988,E2 -4785.988} C_VEL
LIN {X 0,Y 526.248,Z 514.704,A -85,B 0,C 180,E1 -4786.249,E2 -4786.249} C_VEL
LIN {X 0,Y 523.73,Z 501.928,A -85,B 0,C 180,E1 -4786.593,E2 -4786.593} C_VEL
LIN {X 0,Y 523.886,Z 492.105,A -85,B 0,C 180,E1 -4789.595,E2 -4789.595} C_VEL
LIN {X 0,Y 524.022,Z 481.537,A -85,B 0,C 180,E1 -4792.888,E2 -4792.888} C_VEL
LIN {X 0,Y 524.209,Z 472.752,A -85,B 0,C 180,E1 -4795.741,E2 -4795.741} C_VEL
LIN {X 0,Y 524.415,Z 463.458,A -85,B 0,C 180,E1 -4798.845,E2 -4798.845} C_VEL
LIN {X 0,Y 524.641,Z 455.796,A -85,B 0,C 180,E1 -4801.495,E2 -4801.495} C_VEL
LIN {X 0,Y 524.894,Z 446.957,A -85,B 0,C 180,E1 -4804.683,E2 -4804.683} C_VEL
LIN {X 0,Y 525.173,Z 439.63,A -85,B 0,C 180,E1 -4807.442,E2 -4807.442} C_VEL
LIN {X 0,Y 525.088,Z 435.474,A -85,B 0,C 180,E1 -4809.077,E2 -4809.077} C_VEL
LIN {X 0,Y 523.965,Z 428.846,A -85,B 0,C 180,E1 -4811.892,E2 -4811.892} C_VEL
LIN {X 0,Y 523.952,Z 428.846,A -85,B 0,C 180,E1 -4815.308,E2 -4815.308} C_VEL
LIN {X 0,Y 523.957,Z 428.843,A -85,B 0,C 180,E1 -4818.688,E2 -4818.688} C_VEL
LIN {X 0,Y 523.912,Z 428.853,A -85,B 0,C 180,E1 -4821.898,E2 -4821.898} C_VEL
LIN {X 0,Y 523.93,Z 428.849,A -85,B 0,C 180,E1 -4824.909,E2 -4824.909} C_VEL
LIN {X 0,Y 523.938,Z 428.846,A -85,B 0,C 180,E1 -4827.678,E2 -4827.678} C_VEL
LIN {X 0,Y 523.964,Z 428.843,A -85,B 0,C 180,E1 -4830.673,E2 -4830.673} C_VEL
LIN {X 0,Y 523.972,Z 428.842,A -85,B 0,C 180,E1 -4833.729,E2 -4833.729} C_VEL
LIN {X 0,Y 523.93,Z 428.847,A -85,B 0,C 180,E1 -4836.271,E2 -4836.271} C_VEL
LIN {X 0,Y 523.941,Z 428.847,A -85,B 0,C 180,E1 -4838.767,E2 -4838.767} C_VEL
LIN {X 0,Y 523.948,Z 428.847,A -85,B 0,C 180,E1 -4841.221,E2 -4841.221} C_VEL
LIN {X 0,Y 523.935,Z 428.849,A -85,B 0,C 180,E1 -4843.639,E2 -4843.639} C_VEL
LIN {X 0,Y 523.933,Z 428.846,A -85,B 0,C 180,E1 -4846.028,E2 -4846.028} C_VEL
LIN {X 0,Y 524.005,Z 428.839,A -85,B 0,C 180,E1 -4848.394,E2 -4848.394} C_VEL
LIN {X 0,Y 524.002,Z 428.838,A -85,B 0,C 180,E1 -4851.516,E2 -4851.516} C_VEL
LIN {X 0,Y 524.079,Z 428.83,A -85,B 0,C 180,E1 -4854.614,E2 -4854.614} C_VEL
LIN {X 0,Y 524.106,Z 428.828,A -85,B 0,C 180,E1 -4857.695,E2 -4857.695} C_VEL
LIN {X 0,Y 524.118,Z 428.824,A -85,B 0,C 180,E1 -4860.768,E2 -4860.768} C_VEL
LIN {X 0,Y 524.071,Z 428.833,A -85,B 0,C 180,E1 -4863.075,E2 -4863.075} C_VEL
LIN {X 0,Y 524.047,Z 428.834,A -85,B 0,C 180,E1 -4866.159,E2 -4866.159} C_VEL
LIN {X 0,Y 523.997,Z 428.838,A -85,B 0,C 180,E1 -4869.262,E2 -4869.262} C_VEL
LIN {X 0,Y 523.996,Z 428.84,A -85,B 0,C 180,E1 -4871.74,E2 -4871.74} C_VEL
LIN {X 0,Y 523.986,Z 428.841,A -85,B 0,C 180,E1 -4875.053,E2 -4875.053} C_VEL
LIN {X 0,Y 523.959,Z 428.845,A -85,B 0,C 180,E1 -4877.969,E2 -4877.969} C_VEL
LIN {X 0,Y 523.967,Z 428.843,A -85,B 0,C 180,E1 -4880.41,E2 -4880.41} C_VEL
LIN {X 0,Y 523.912,Z 428.849,A -85,B 0,C 180,E1 -4882.894,E2 -4882.894} C_VEL
LIN {X 0,Y 523.948,Z 428.846,A -85,B 0,C 180,E1 -4885.419,E2 -4885.419} C_VEL
LIN {X 0,Y 523.965,Z 428.846,A -85,B 0,C 180,E1 -4887.999,E2 -4887.999} C_VEL
LIN {X 0,Y 523.943,Z 428.846,A -85,B 0,C 180,E1 -4890.856,E2 -4890.856} C_VEL
LIN {X 0,Y 523.957,Z 428.845,A -85,B 0,C 180,E1 -4893.735,E2 -4893.735} C_VEL
LIN {X 0,Y 523.918,Z 428.85,A -85,B 0,C 180,E1 -4896.405,E2 -4896.405} C_VEL
LIN {X 0,Y 523.917,Z 428.85,A -85,B 0,C 180,E1 -4899.085,E2 -4899.085} C_VEL
LIN {X 0,Y 523.954,Z 428.845,A -85,B 0,C 180,E1 -4902.119,E2 -4902.119} C_VEL
LIN {X 0,Y 523.955,Z 428.844,A -85,B 0,C 180,E1 -4905.309,E2 -4905.309} C_VEL
LIN {X 0,Y 523.917,Z 428.85,A -85,B 0,C 180,E1 -4906.924,E2 -4906.924} C_VEL
LIN {X 0,Y 523.252,Z 428.933,A -85,B 0,C 180,E1 -4907.565,E2 -4907.565} C_VEL
LIN {X 0,Y 520.416,Z 429.286,A -85,B 0,C 180,E1 -4908.607,E2 -4908.607} C_VEL
LIN {X 0,Y 518.015,Z 429.586,A -85,B 0,C 180,E1 -4909.446,E2 -4909.446} C_VEL
LIN {X 0,Y 516.98,Z 429.715,A -85,B 0,C 180,E1 -4910.094,E2 -4910.094} C_VEL
LIN {X 0,Y 516.892,Z 429.724,A -85,B 0,C 180,E1 -4910.313,E2 -4910.313} C_VEL
LIN {X 0,Y 516.885,Z 429.724,A -85,B 0,C 180,E1 -4913.342,E2 -4913.342} C_VEL
LIN {X 0,Y 516.913,Z 429.722,A -85,B 0,C 180,E1 -4916.122,E2 -4916.122} C_VEL
LIN {X 0,Y 516.894,Z 429.723,A -85,B 0,C 180,E1 -4918.936,E2 -4918.936} C_VEL
LIN {X 0,Y 516.923,Z 429.72,A -85,B 0,C 180,E1 -4921.586,E2 -4921.586} C_VEL
LIN {X 0,Y 516.934,Z 429.719,A -85,B 0,C 180,E1 -4924.212,E2 -4924.212} C_VEL
LIN {X 0,Y 516.868,Z 429.727,A -85,B 0,C 180,E1 -4926.777,E2 -4926.777} C_VEL
LIN {X 0,Y 516.943,Z 429.718,A -85,B 0,C 180,E1 -4929.732,E2 -4929.732} C_VEL
LIN {X 0,Y 516.925,Z 429.719,A -85,B 0,C 180,E1 -4932.596,E2 -4932.596} C_VEL
LIN {X 0,Y 516.946,Z 429.718,A -85,B 0,C 180,E1 -4935.031,E2 -4935.031} C_VEL
LIN {X 0,Y 516.97,Z 429.715,A -85,B 0,C 180,E1 -4938.234,E2 -4938.234} C_VEL
LIN {X 0,Y 516.97,Z 429.718,A -85,B 0,C 180,E1 -4941.4,E2 -4941.4} C_VEL
LIN {X 0,Y 517.028,Z 429.708,A -85,B 0,C 180,E1 -4944.54,E2 -4944.54} C_VEL
LIN {X 0,Y 517.089,Z 429.7,A -85,B 0,C 180,E1 -4947.663,E2 -4947.663} C_VEL
LIN {X 0,Y 517.096,Z 429.699,A -85,B 0,C 180,E1 -4950.779,E2 -4950.779} C_VEL
LIN {X 0,Y 517.016,Z 429.709,A -85,B 0,C 180,E1 -4953.117,E2 -4953.117} C_VEL
LIN {X 0,Y 517.016,Z 429.71,A -85,B 0,C 180,E1 -4956.243,E2 -4956.243} C_VEL
LIN {X 0,Y 516.954,Z 429.719,A -85,B 0,C 180,E1 -4959.389,E2 -4959.389} C_VEL
LIN {X 0,Y 516.957,Z 429.718,A -85,B 0,C 180,E1 -4961.807,E2 -4961.807} C_VEL
LIN {X 0,Y 516.948,Z 429.718,A -85,B 0,C 180,E1 -4965.146,E2 -4965.146} C_VEL
LIN {X 0,Y 516.928,Z 429.718,A -85,B 0,C 180,E1 -4968.222,E2 -4968.222} C_VEL
LIN {X 0,Y 516.915,Z 429.722,A -85,B 0,C 180,E1 -4970.701,E2 -4970.701} C_VEL
LIN {X 0,Y 516.914,Z 429.722,A -85,B 0,C 180,E1 -4974.071,E2 -4974.071} C_VEL
LIN {X 0,Y 516.929,Z 429.719,A -85,B 0,C 180,E1 -4976.657,E2 -4976.657} C_VEL
LIN {X 0,Y 516.913,Z 429.722,A -85,B 0,C 180,E1 -4979.523,E2 -4979.523} C_VEL
LIN {X 0,Y 516.897,Z 429.725,A -85,B 0,C 180,E1 -4982.543,E2 -4982.543} C_VEL
LIN {X 0,Y 516.753,Z 429.746,A -85,B 0,C 180,E1 -4985.311,E2 -4985.311} C_VEL
LIN {X 0,Y 516.58,Z 429.767,A -85,B 0,C 180,E1 -4986.77,E2 -4986.77} C_VEL
LIN {X 0,Y 516.484,Z 430.237,A -85,B 0,C 180,E1 -4987.886,E2 -4987.886} C_VEL
LIN {X 0,Y 516.445,Z 433.046,A -85,B 0,C 180,E1 -4990.783,E2 -4990.783} C_VEL
LIN {X 0,Y 516.435,Z 436.1,A -85,B 0,C 180,E1 -4993.95,E2 -4993.95} C_VEL
LIN {X 0,Y 516.384,Z 439.37,A -85,B 0,C 180,E1 -4997.301,E2 -4997.301} C_VEL
LIN {X 0,Y 516.313,Z 442.253,A -85,B 0,C 180,E1 -5000.226,E2 -5000.226} C_VEL
LIN {X 0,Y 516.25,Z 445.219,A -85,B 0,C 180,E1 -5003.202,E2 -5003.202} C_VEL
LIN {X 0,Y 516.253,Z 447.31,A -85,B 0,C 180,E1 -5005.295,E2 -5005.295} C_VEL
LIN {X 0,Y 519.436,Z 461.257,A -85,B 0,C 180,E1 -5005.734,E2 -5005.734} C_VEL
LIN {X 0,Y 519.165,Z 475.61,A -85,B 0,C 180,E1 -5006.229,E2 -5006.229} C_VEL
LIN {X 0,Y 518.783,Z 489.343,A -85,B 0,C 180,E1 -5006.876,E2 -5006.876} C_VEL
LIN {X 0,Y 518.384,Z 501.66,A -85,B 0,C 180,E1 -5007.62,E2 -5007.62} C_VEL
LIN {X 0,Y 517.99,Z 512.868,A -85,B 0,C 180,E1 -5008.454,E2 -5008.454} C_VEL
